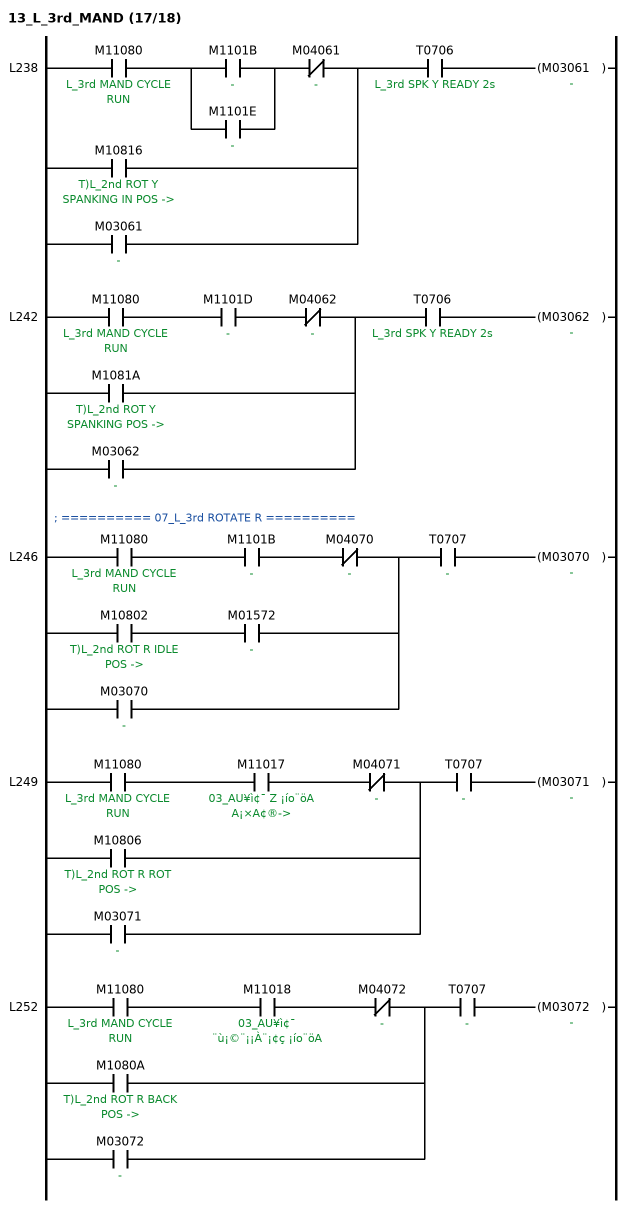
[picture p96: 13_L_3rd_MAND rungs L238-L252]
; L238
LOAD      M11080	// L_3rd MAND CYCLE RUN
LOAD      M1101B	// -
OR        M1101E	// -
AND LOAD
AND NOT   M04061	// -
OR        M10816	// T)L_2nd ROT Y SPANKING IN POS ->
OR        M03061	// -
AND       T0706	// L_3rd SPK Y READY 2s
OUT       M03061	// -
; L242
LOAD      M11080	// L_3rd MAND CYCLE RUN
AND       M1101D	// -
AND NOT   M04062	// -
OR        M1081A	// T)L_2nd ROT Y SPANKING POS ->
OR        M03062	// -
AND       T0706	// L_3rd SPK Y READY 2s
OUT       M03062	// -
// ========== 07_L_3rd ROTATE R ==========
; L246
LOAD      M11080	// L_3rd MAND CYCLE RUN
AND       M1101B	// -
AND NOT   M04070	// -
LOAD      M10802	// T)L_2nd ROT R IDLE POS ->
AND       M01572	// -
OR LOAD
OR        M03070	// -
AND       T0707	// -
OUT       M03070	// -
; L249
LOAD      M11080	// L_3rd MAND CYCLE RUN
AND       M11017	// 03_AU¥ì¢¯ Z ¡ío¨öA A¡×A¢®->
AND NOT   M04071	// -
OR        M10806	// T)L_2nd ROT R ROT POS ->
OR        M03071	// -
AND       T0707	// -
OUT       M03071	// -
; L252
LOAD      M11080	// L_3rd MAND CYCLE RUN
AND       M11018	// 03_AU¥ì¢¯ ¨ù¡©¨¡¡À¨¡¢ç ¡ío¨öA
AND NOT   M04072	// -
OR        M1080A	// T)L_2nd ROT R BACK POS ->
OR        M03072	// -
AND       T0707	// -
OUT       M03072	// -

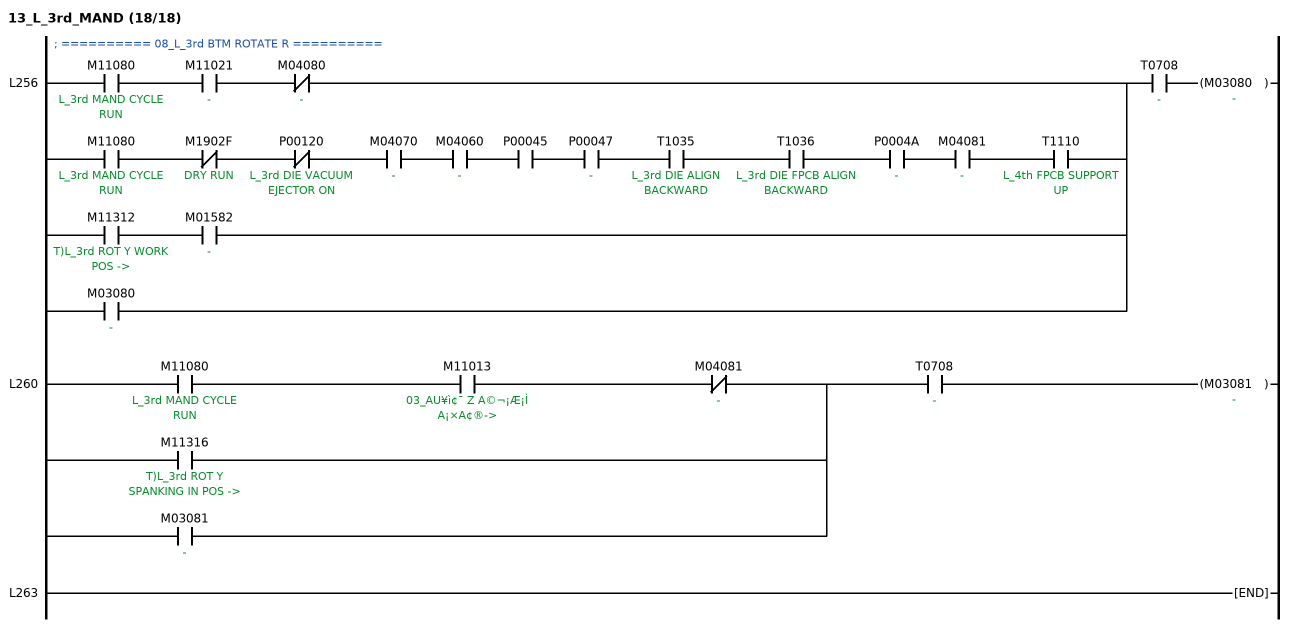
// ========== 08_L_3rd BTM ROTATE R ==========
; L256
LOAD      M11080	// L_3rd MAND CYCLE RUN
AND       M11021	// -
AND NOT   M04080	// -
LOAD      M11080	// L_3rd MAND CYCLE RUN
AND NOT   M1902F	// DRY RUN
AND NOT   P00120	// L_3rd DIE VACUUM EJECTOR ON
AND       M04070	// -
AND       M04060	// -
AND       P00045
AND       P00047	// -
AND       T1035	// L_3rd DIE ALIGN BACKWARD
AND       T1036	// L_3rd DIE FPCB ALIGN BACKWARD
AND       P0004A	// -
AND       M04081	// -
AND       T1110	// L_4th FPCB SUPPORT UP
OR LOAD
LOAD      M11312	// T)L_3rd ROT Y WORK POS ->
AND       M01582	// -
OR LOAD
OR        M03080	// -
AND       T0708	// -
OUT       M03080	// -
; L260
LOAD      M11080	// L_3rd MAND CYCLE RUN
AND       M11013	// 03_AU¥ì¢¯ Z A©¬¡Æ¡Ì A¡×A¢®->
AND NOT   M04081	// -
OR        M11316	// T)L_3rd ROT Y SPANKING IN POS ->
OR        M03081	// -
AND       T0708	// -
OUT       M03081	// -
; L263
END

PROGRAM 14_L_TOOL (task: ¨ö¨¬A¥ì CA¡¤I¡¾¡¿¡¤¡Í)

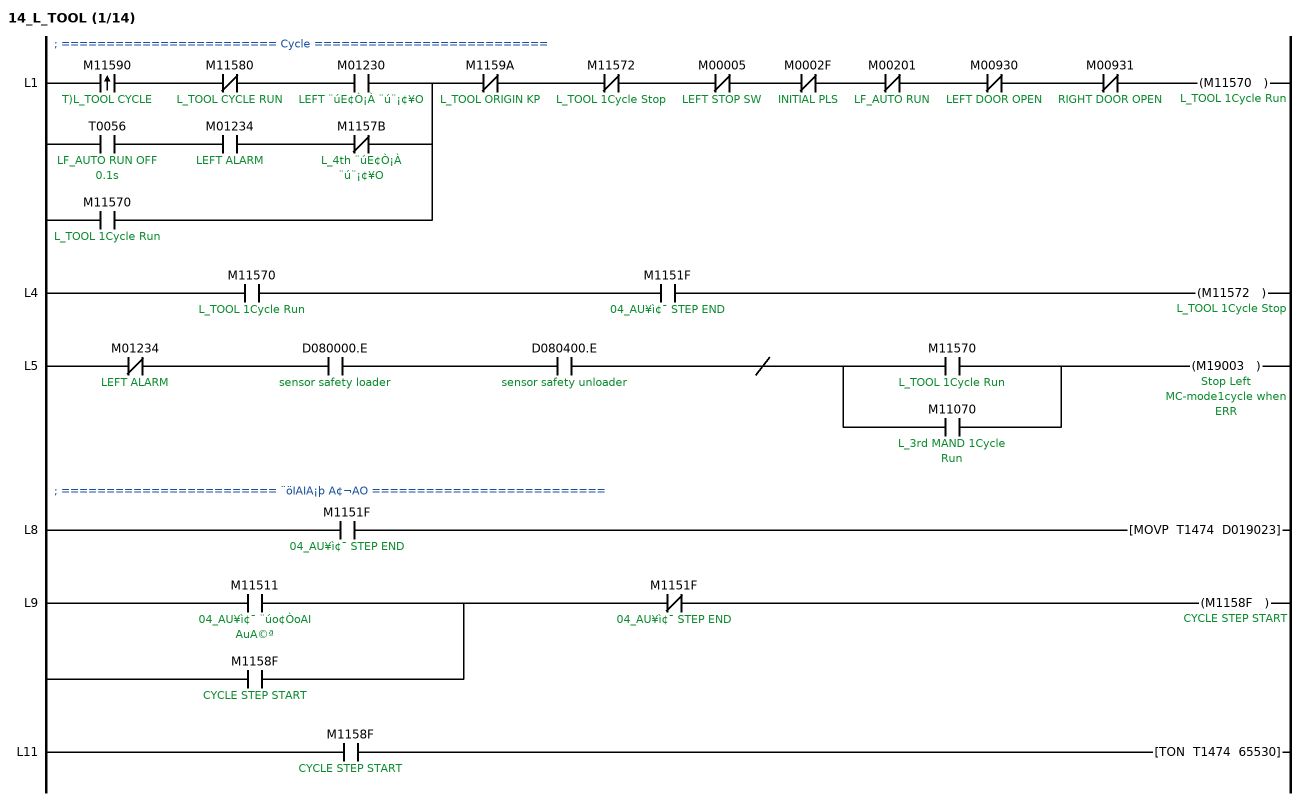
// ======================== Cycle ==========================
; L1
LOADP     M11590	// T)L_TOOL CYCLE
AND NOT   M11580	// L_TOOL CYCLE RUN
AND       M01230	// LEFT ¨úE¢Ò¡À ¨ú¨¡¢¥O
LOAD      T0056	// LF_AUTO RUN OFF 0.1s
AND       M01234	// LEFT ALARM
AND NOT   M1157B	// L_4th ¨úE¢Ò¡À ¨ú¨¡¢¥O
OR LOAD
OR        M11570	// L_TOOL 1Cycle Run
AND NOT   M1159A	// L_TOOL ORIGIN KP
AND NOT   M11572	// L_TOOL 1Cycle Stop
AND NOT   M00005	// LEFT STOP SW
AND NOT   M0002F	// INITIAL PLS
AND NOT   M00201	// LF_AUTO RUN
AND NOT   M00930	// LEFT DOOR OPEN
AND NOT   M00931	// RIGHT DOOR OPEN
OUT       M11570	// L_TOOL 1Cycle Run
; L4
LOAD      M11570	// L_TOOL 1Cycle Run
AND       M1151F	// 04_AU¥ì¢¯ STEP END
OUT       M11572	// L_TOOL 1Cycle Stop
; L5
LOAD NOT  M01234	// LEFT ALARM
AND       D080000.E	// sensor safety loader
AND       D080400.E	// sensor safety unloader
NOT
LOAD      M11570	// L_TOOL 1Cycle Run
OR        M11070	// L_3rd MAND 1Cycle Run
AND LOAD
OUT       M19003	// Stop Left MC-mode1cycle when ERR
// ======================== ¨öIAIA¡þ A¢¬AO ==========================
; L8
LOAD      M1151F	// 04_AU¥ì¢¯ STEP END
MOVP      T1474 D019023
; L9
LOAD      M11511	// 04_AU¥ì¢¯ ¨úo¢ÒoAI AuA©ª
OR        M1158F	// CYCLE STEP START
AND NOT   M1151F	// 04_AU¥ì¢¯ STEP END
OUT       M1158F	// CYCLE STEP START
; L11
LOAD      M1158F	// CYCLE STEP START
TON       T1474 65530

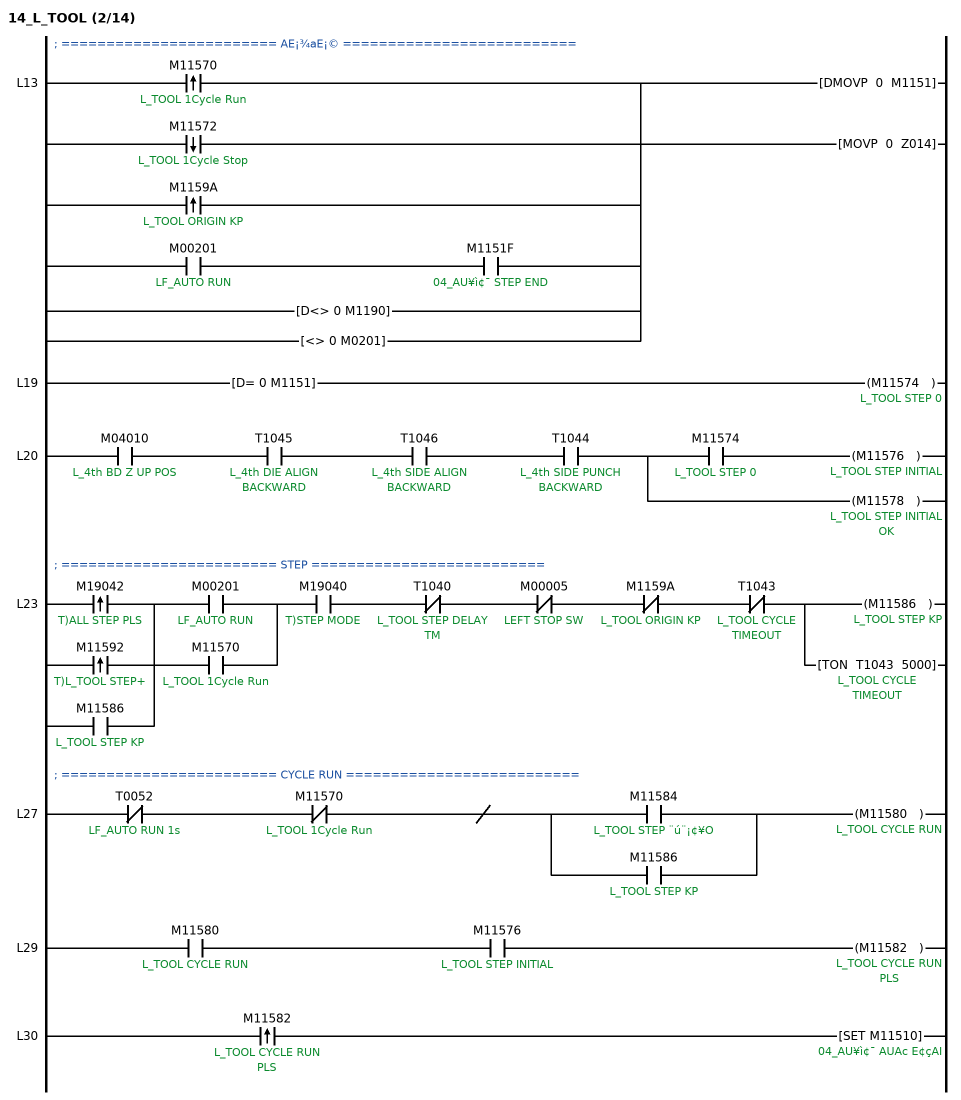
// ======================== AE¡¾aE¡© ==========================
; L13
LOADP     M11570	// L_TOOL 1Cycle Run
ORN       M11572	// L_TOOL 1Cycle Stop
ORP       M1159A	// L_TOOL ORIGIN KP
LOAD      M00201	// LF_AUTO RUN
AND       M1151F	// 04_AU¥ì¢¯ STEP END
OR LOAD
ORD<>     0 M1190
OR<>      0 M0201
DMOVP     0 M1151
MOVP      0 Z014
; L19
LOADD=    0 M1151
OUT       M11574	// L_TOOL STEP 0
; L20
LOAD      M04010	// L_4th BD Z UP POS
AND       T1045	// L_4th DIE ALIGN BACKWARD
AND       T1046	// L_4th SIDE ALIGN BACKWARD
AND       T1044	// L_4th SIDE PUNCH BACKWARD
MPUSH
AND       M11574	// L_TOOL STEP 0
OUT       M11576	// L_TOOL STEP INITIAL
MPOP
OUT       M11578	// L_TOOL STEP INITIAL OK
// ======================== STEP ==========================
; L23
LOADP     M19042	// T)ALL STEP PLS
ORP       M11592	// T)L_TOOL STEP+
OR        M11586	// L_TOOL STEP KP
LOAD      M00201	// LF_AUTO RUN
OR        M11570	// L_TOOL 1Cycle Run
AND LOAD
AND       M19040	// T)STEP MODE
AND NOT   T1040	// L_TOOL STEP DELAY TM
AND NOT   M00005	// LEFT STOP SW
AND NOT   M1159A	// L_TOOL ORIGIN KP
AND NOT   T1043	// L_TOOL CYCLE TIMEOUT
OUT       M11586	// L_TOOL STEP KP
TON       T1043 5000	// L_TOOL CYCLE TIMEOUT
// ======================== CYCLE RUN ==========================
; L27
LOAD NOT  T0052	// LF_AUTO RUN 1s
AND NOT   M11570	// L_TOOL 1Cycle Run
NOT
LOAD      M11584	// L_TOOL STEP ¨ú¨¡¢¥O
OR        M11586	// L_TOOL STEP KP
AND LOAD
OUT       M11580	// L_TOOL CYCLE RUN
; L29
LOAD      M11580	// L_TOOL CYCLE RUN
AND       M11576	// L_TOOL STEP INITIAL
OUT       M11582	// L_TOOL CYCLE RUN PLS
; L30
LOADP     M11582	// L_TOOL CYCLE RUN PLS
SET       M11510	// 04_AU¥ì¢¯ AUAc E¢çAI

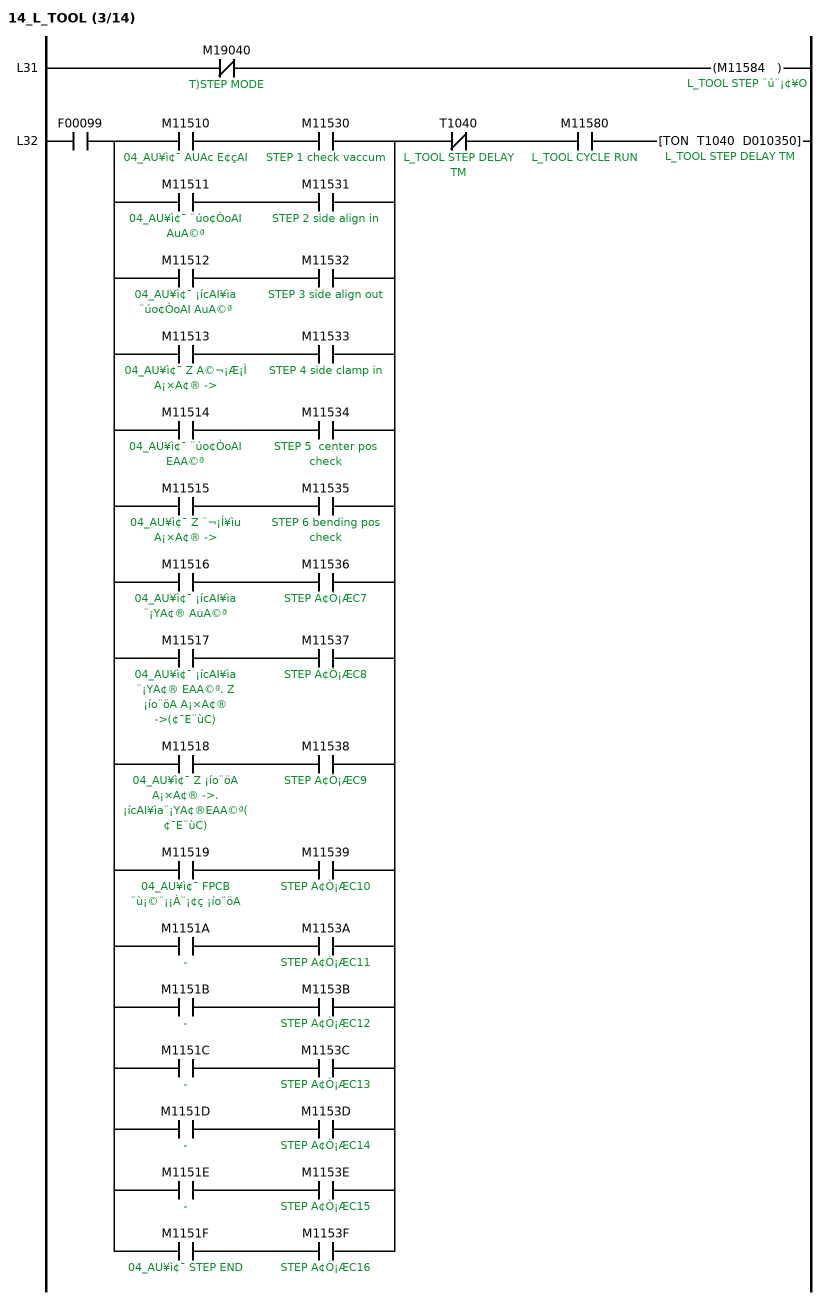
; L31
LOAD NOT  M19040	// T)STEP MODE
OUT       M11584	// L_TOOL STEP ¨ú¨¡¢¥O
; L32
LOAD      F00099
LOAD      M11510	// 04_AU¥ì¢¯ AUAc E¢çAI
AND       M11530	// STEP 1 check vaccum
LOAD      M11511	// 04_AU¥ì¢¯ ¨úo¢ÒoAI AuA©ª
AND       M11531	// STEP 2 side align in
OR LOAD
LOAD      M11512	// 04_AU¥ì¢¯ ¡ícAI¥ìa ¨úo¢ÒoAI AuA©ª
AND       M11532	// STEP 3 side align out
OR LOAD
LOAD      M11513	// 04_AU¥ì¢¯ Z A©¬¡Æ¡Ì A¡×A¢® ->
AND       M11533	// STEP 4 side clamp in
OR LOAD
LOAD      M11514	// 04_AU¥ì¢¯ ¨úo¢ÒoAI EAA©ª
AND       M11534	// STEP 5  center pos check
OR LOAD
LOAD      M11515	// 04_AU¥ì¢¯ Z ¨¬¡Í¥ìu A¡×A¢® ->
AND       M11535	// STEP 6 bending pos check
OR LOAD
LOAD      M11516	// 04_AU¥ì¢¯ ¡ícAI¥ìa ¨¡YA¢® AuA©ª
AND       M11536	// STEP A¢Ò¡ÆC7
OR LOAD
LOAD      M11517	// 04_AU¥ì¢¯ ¡ícAI¥ìa ¨¡YA¢® EAA©ª. Z ¡ío¨öA A¡×A¢® ->(¢¯E¨ùC)
AND       M11537	// STEP A¢Ò¡ÆC8
OR LOAD
LOAD      M11518	// 04_AU¥ì¢¯ Z ¡ío¨öA A¡×A¢® ->. ¡ícAI¥ìa¨¡YA¢®EAA©ª(¢¯E¨ùC)
AND       M11538	// STEP A¢Ò¡ÆC9
OR LOAD
LOAD      M11519	// 04_AU¥ì¢¯ FPCB ¨ù¡©¨¡¡À¨¡¢ç ¡ío¨öA
AND       M11539	// STEP A¢Ò¡ÆC10
OR LOAD
LOAD      M1151A	// -
AND       M1153A	// STEP A¢Ò¡ÆC11
OR LOAD
LOAD      M1151B	// -
AND       M1153B	// STEP A¢Ò¡ÆC12
OR LOAD
LOAD      M1151C	// -
AND       M1153C	// STEP A¢Ò¡ÆC13
OR LOAD
LOAD      M1151D	// -
AND       M1153D	// STEP A¢Ò¡ÆC14
OR LOAD
LOAD      M1151E	// -
AND       M1153E	// STEP A¢Ò¡ÆC15
OR LOAD
LOAD      M1151F	// 04_AU¥ì¢¯ STEP END
AND       M1153F	// STEP A¢Ò¡ÆC16
OR LOAD
AND LOAD
AND NOT   T1040	// L_TOOL STEP DELAY TM
AND       M11580	// L_TOOL CYCLE RUN
TON       T1040 D010350	// L_TOOL STEP DELAY TM

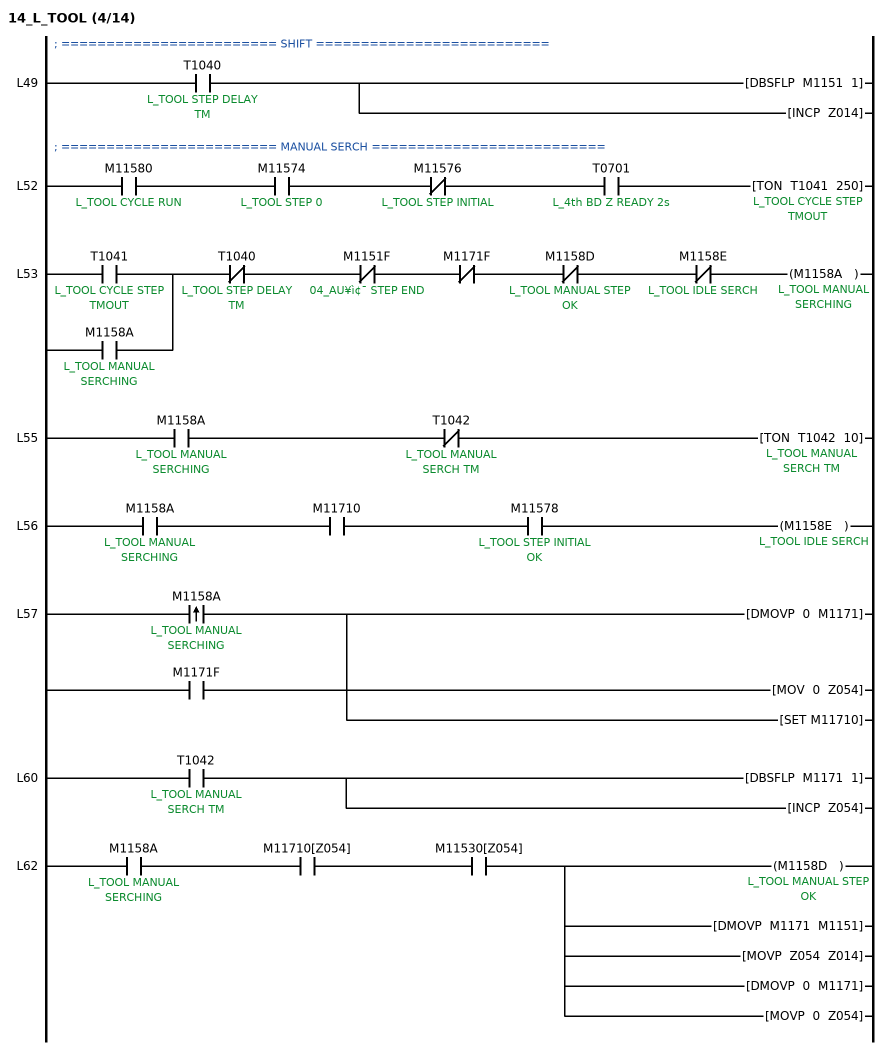
// ======================== SHIFT ==========================
; L49
LOAD      T1040	// L_TOOL STEP DELAY TM
DBSFLP    M1151 1
INCP      Z014
// ======================== MANUAL SERCH ==========================
; L52
LOAD      M11580	// L_TOOL CYCLE RUN
AND       M11574	// L_TOOL STEP 0
AND NOT   M11576	// L_TOOL STEP INITIAL
AND       T0701	// L_4th BD Z READY 2s
TON       T1041 250	// L_TOOL CYCLE STEP TMOUT
; L53
LOAD      T1041	// L_TOOL CYCLE STEP TMOUT
OR        M1158A	// L_TOOL MANUAL SERCHING
AND NOT   T1040	// L_TOOL STEP DELAY TM
AND NOT   M1151F	// 04_AU¥ì¢¯ STEP END
AND NOT   M1171F
AND NOT   M1158D	// L_TOOL MANUAL STEP OK
AND NOT   M1158E	// L_TOOL IDLE SERCH
OUT       M1158A	// L_TOOL MANUAL SERCHING
; L55
LOAD      M1158A	// L_TOOL MANUAL SERCHING
AND NOT   T1042	// L_TOOL MANUAL SERCH TM
TON       T1042 10	// L_TOOL MANUAL SERCH TM
; L56
LOAD      M1158A	// L_TOOL MANUAL SERCHING
AND       M11710
AND       M11578	// L_TOOL STEP INITIAL OK
OUT       M1158E	// L_TOOL IDLE SERCH
; L57
LOADP     M1158A	// L_TOOL MANUAL SERCHING
OR        M1171F
DMOVP     0 M1171
MOV       0 Z054
SET       M11710
; L60
LOAD      T1042	// L_TOOL MANUAL SERCH TM
DBSFLP    M1171 1
INCP      Z054
; L62
LOAD      M1158A	// L_TOOL MANUAL SERCHING
AND       M11710[Z054]
AND       M11530[Z054]
OUT       M1158D	// L_TOOL MANUAL STEP OK
DMOVP     M1171 M1151
MOVP      Z054 Z014
DMOVP     0 M1171
MOVP      0 Z054

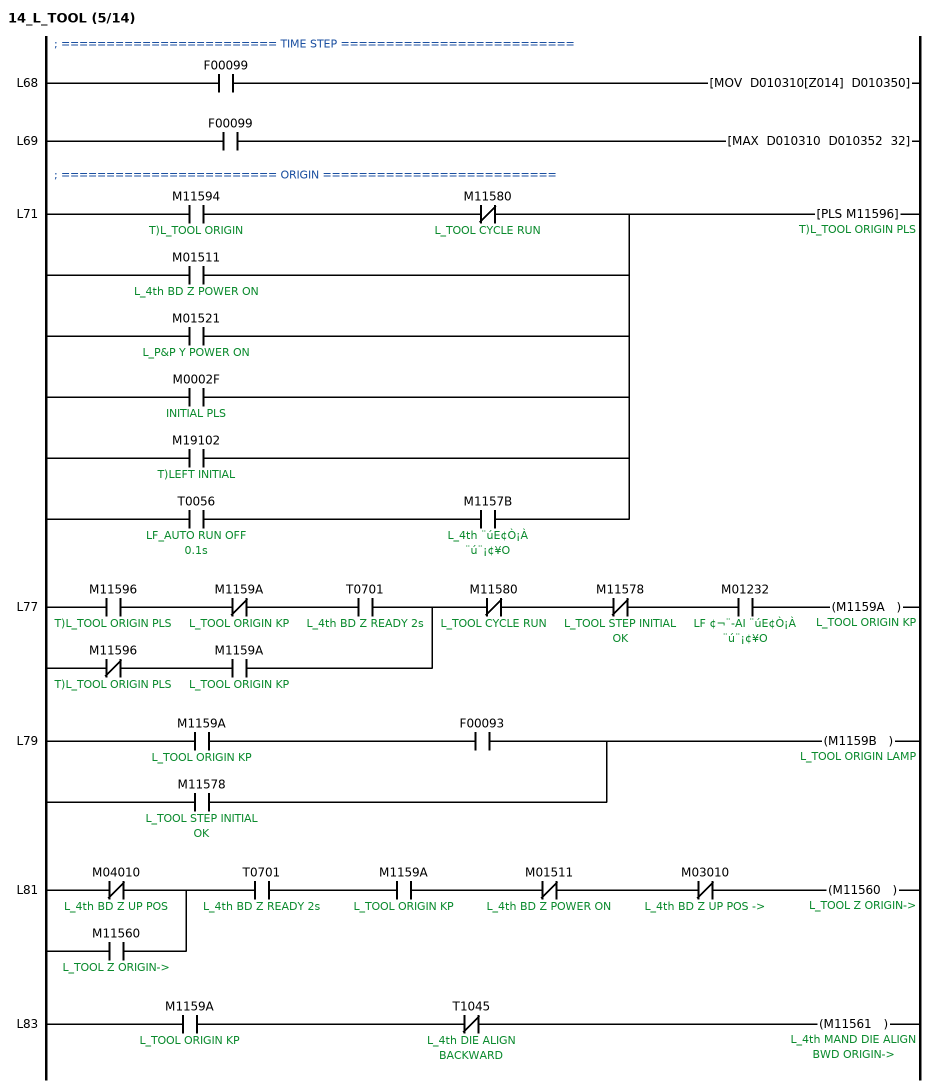
// ======================== TIME STEP ==========================
; L68
LOAD      F00099
MOV       D010310[Z014] D010350
; L69
LOAD      F00099
MAX       D010310 D010352 32
// ======================== ORIGIN ==========================
; L71
LOAD      M11594	// T)L_TOOL ORIGIN
AND NOT   M11580	// L_TOOL CYCLE RUN
OR        M01511	// L_4th BD Z POWER ON
OR        M01521	// L_P&P Y POWER ON
OR        M0002F	// INITIAL PLS
OR        M19102	// T)LEFT INITIAL
LOAD      T0056	// LF_AUTO RUN OFF 0.1s
AND       M1157B	// L_4th ¨úE¢Ò¡À ¨ú¨¡¢¥O
OR LOAD
OUTP      M11596	// T)L_TOOL ORIGIN PLS
; L77
LOAD      M11596	// T)L_TOOL ORIGIN PLS
AND NOT   M1159A	// L_TOOL ORIGIN KP
AND       T0701	// L_4th BD Z READY 2s
LOAD NOT  M11596	// T)L_TOOL ORIGIN PLS
AND       M1159A	// L_TOOL ORIGIN KP
OR LOAD
AND NOT   M11580	// L_TOOL CYCLE RUN
AND NOT   M11578	// L_TOOL STEP INITIAL OK
AND       M01232	// LF ¢¬¨­AI ¨úE¢Ò¡À ¨ú¨¡¢¥O
OUT       M1159A	// L_TOOL ORIGIN KP
; L79
LOAD      M1159A	// L_TOOL ORIGIN KP
AND       F00093
OR        M11578	// L_TOOL STEP INITIAL OK
OUT       M1159B	// L_TOOL ORIGIN LAMP
; L81
LOAD NOT  M04010	// L_4th BD Z UP POS
OR        M11560	// L_TOOL Z ORIGIN->
AND       T0701	// L_4th BD Z READY 2s
AND       M1159A	// L_TOOL ORIGIN KP
AND NOT   M01511	// L_4th BD Z POWER ON
AND NOT   M03010	// L_4th BD Z UP POS ->
OUT       M11560	// L_TOOL Z ORIGIN->
; L83
LOAD      M1159A	// L_TOOL ORIGIN KP
AND NOT   T1045	// L_4th DIE ALIGN BACKWARD
OUT       M11561	// L_4th MAND DIE ALIGN BWD ORIGIN->

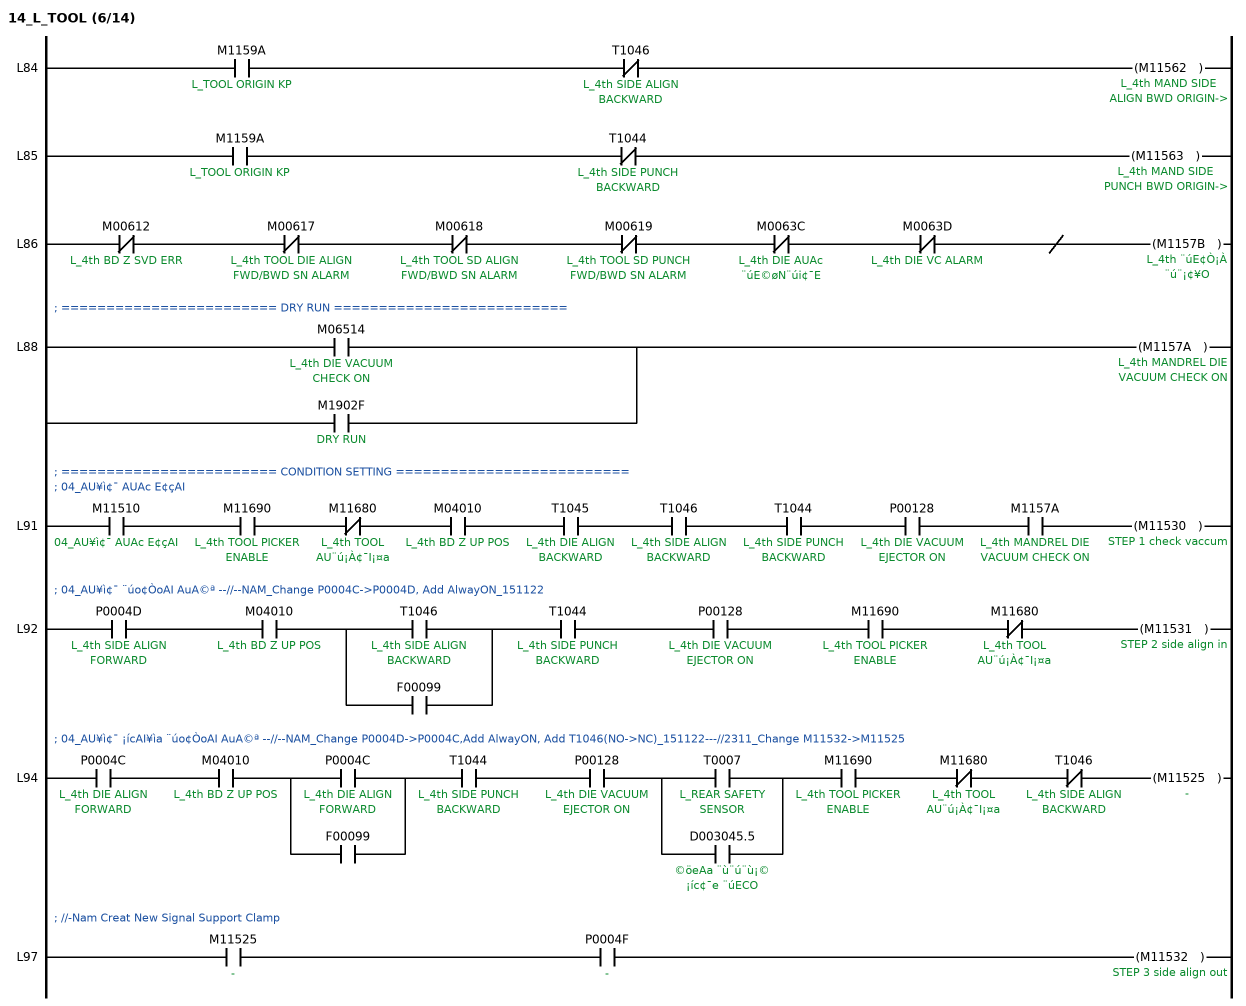
; L84
LOAD      M1159A	// L_TOOL ORIGIN KP
AND NOT   T1046	// L_4th SIDE ALIGN BACKWARD
OUT       M11562	// L_4th MAND SIDE ALIGN BWD ORIGIN->
; L85
LOAD      M1159A	// L_TOOL ORIGIN KP
AND NOT   T1044	// L_4th SIDE PUNCH BACKWARD
OUT       M11563	// L_4th MAND SIDE PUNCH BWD ORIGIN->
; L86
LOAD NOT  M00612	// L_4th BD Z SVD ERR
AND NOT   M00617	// L_4th TOOL DIE ALIGN FWD/BWD SN ALARM
AND NOT   M00618	// L_4th TOOL SD ALIGN FWD/BWD SN ALARM
AND NOT   M00619	// L_4th TOOL SD PUNCH FWD/BWD SN ALARM
AND NOT   M0063C	// L_4th DIE AUAc ¨úE©øN¨úi¢¯E
AND NOT   M0063D	// L_4th DIE VC ALARM
NOT
OUT       M1157B	// L_4th ¨úE¢Ò¡À ¨ú¨¡¢¥O
// ======================== DRY RUN ==========================
; L88
LOAD      M06514	// L_4th DIE VACUUM CHECK ON
OR        M1902F	// DRY RUN
OUT       M1157A	// L_4th MANDREL DIE VACUUM CHECK ON
// ======================== CONDITION SETTING ==========================
; L91
LOAD      M11510	// 04_AU¥ì¢¯ AUAc E¢çAI
AND       M11690	// L_4th TOOL PICKER ENABLE
AND NOT   M11680	// L_4th TOOL AU¨ú¡À¢¯I¡¤a
AND       M04010	// L_4th BD Z UP POS
AND       T1045	// L_4th DIE ALIGN BACKWARD
AND       T1046	// L_4th SIDE ALIGN BACKWARD
AND       T1044	// L_4th SIDE PUNCH BACKWARD
AND       P00128	// L_4th DIE VACUUM EJECTOR ON
AND       M1157A	// L_4th MANDREL DIE VACUUM CHECK ON
OUT       M11530	// STEP 1 check vaccum
// output comment: 04_AU¥ì¢¯ AUAc E¢çAI
; L92
LOAD      P0004D	// L_4th SIDE ALIGN FORWARD
AND       M04010	// L_4th BD Z UP POS
LOAD      T1046	// L_4th SIDE ALIGN BACKWARD
OR        F00099
AND LOAD
AND       T1044	// L_4th SIDE PUNCH BACKWARD
AND       P00128	// L_4th DIE VACUUM EJECTOR ON
AND       M11690	// L_4th TOOL PICKER ENABLE
AND NOT   M11680	// L_4th TOOL AU¨ú¡À¢¯I¡¤a
OUT       M11531	// STEP 2 side align in
// output comment: 04_AU¥ì¢¯ ¨úo¢ÒoAI AuA©ª --//--NAM_Change P0004C->P0004D, Add AlwayON_151122
; L94
LOAD      P0004C	// L_4th DIE ALIGN FORWARD
AND       M04010	// L_4th BD Z UP POS
LOAD      P0004C	// L_4th DIE ALIGN FORWARD
OR        F00099
AND LOAD
AND       T1044	// L_4th SIDE PUNCH BACKWARD
AND       P00128	// L_4th DIE VACUUM EJECTOR ON
LOAD      T0007	// L_REAR SAFETY SENSOR
OR        D003045.5	// ©öeAa ¨ù¨ú¨ù¡© ¡íc¢¯e ¨úECO
AND LOAD
AND       M11690	// L_4th TOOL PICKER ENABLE
AND NOT   M11680	// L_4th TOOL AU¨ú¡À¢¯I¡¤a
AND NOT   T1046	// L_4th SIDE ALIGN BACKWARD
OUT       M11525	// -
// output comment: 04_AU¥ì¢¯ ¡ícAI¥ìa ¨úo¢ÒoAI AuA©ª --//--NAM_Change P0004D->P0004C,Add AlwayON, Add T1046(NO->NC)_151122---//2311_Change M11532->M11525
// //-Nam Creat New Signal Support Clamp
; L97
LOAD      M11525	// -
AND       P0004F	// -
OUT       M11532	// STEP 3 side align out

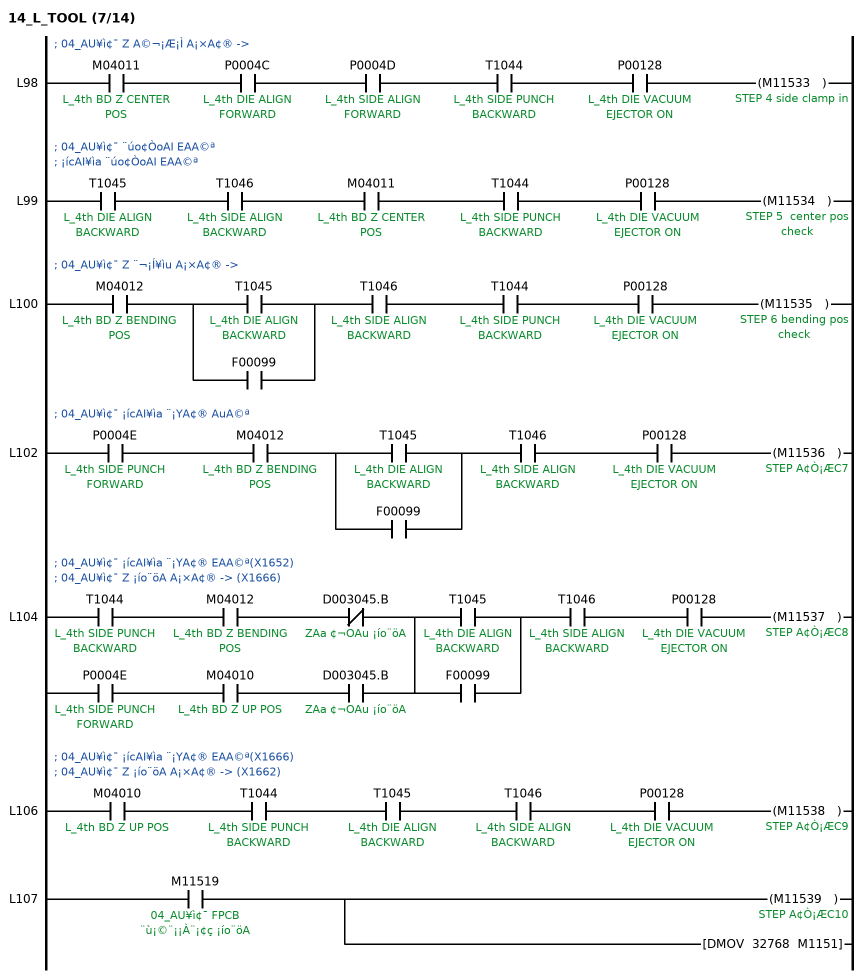
; L98
LOAD      M04011	// L_4th BD Z CENTER POS
AND       P0004C	// L_4th DIE ALIGN FORWARD
AND       P0004D	// L_4th SIDE ALIGN FORWARD
AND       T1044	// L_4th SIDE PUNCH BACKWARD
AND       P00128	// L_4th DIE VACUUM EJECTOR ON
OUT       M11533	// STEP 4 side clamp in
// output comment: 04_AU¥ì¢¯ Z A©¬¡Æ¡Ì A¡×A¢® ->
; L99
LOAD      T1045	// L_4th DIE ALIGN BACKWARD
AND       T1046	// L_4th SIDE ALIGN BACKWARD
AND       M04011	// L_4th BD Z CENTER POS
AND       T1044	// L_4th SIDE PUNCH BACKWARD
AND       P00128	// L_4th DIE VACUUM EJECTOR ON
OUT       M11534	// STEP 5  center pos check
// output comment: 04_AU¥ì¢¯ ¨úo¢ÒoAI EAA©ª ¡ícAI¥ìa ¨úo¢ÒoAI EAA©ª
; L100
LOAD      M04012	// L_4th BD Z BENDING POS
LOAD      T1045	// L_4th DIE ALIGN BACKWARD
OR        F00099
AND LOAD
AND       T1046	// L_4th SIDE ALIGN BACKWARD
AND       T1044	// L_4th SIDE PUNCH BACKWARD
AND       P00128	// L_4th DIE VACUUM EJECTOR ON
OUT       M11535	// STEP 6 bending pos check
// output comment: 04_AU¥ì¢¯ Z ¨¬¡Í¥ìu A¡×A¢® ->
; L102
LOAD      P0004E	// L_4th SIDE PUNCH FORWARD
AND       M04012	// L_4th BD Z BENDING POS
LOAD      T1045	// L_4th DIE ALIGN BACKWARD
OR        F00099
AND LOAD
AND       T1046	// L_4th SIDE ALIGN BACKWARD
AND       P00128	// L_4th DIE VACUUM EJECTOR ON
OUT       M11536	// STEP A¢Ò¡ÆC7
// output comment: 04_AU¥ì¢¯ ¡ícAI¥ìa ¨¡YA¢® AuA©ª
; L104
LOAD      T1044	// L_4th SIDE PUNCH BACKWARD
AND       M04012	// L_4th BD Z BENDING POS
AND NOT   D003045.B	// ZAa ¢¬OAu ¡ío¨öA
LOAD      P0004E	// L_4th SIDE PUNCH FORWARD
AND       M04010	// L_4th BD Z UP POS
AND       D003045.B	// ZAa ¢¬OAu ¡ío¨öA
OR LOAD
LOAD      T1045	// L_4th DIE ALIGN BACKWARD
OR        F00099
AND LOAD
AND       T1046	// L_4th SIDE ALIGN BACKWARD
AND       P00128	// L_4th DIE VACUUM EJECTOR ON
OUT       M11537	// STEP A¢Ò¡ÆC8
// output comment: 04_AU¥ì¢¯ ¡ícAI¥ìa ¨¡YA¢® EAA©ª(X1652) 04_AU¥ì¢¯ Z ¡ío¨öA A¡×A¢® -> (X1666)
; L106
LOAD      M04010	// L_4th BD Z UP POS
AND       T1044	// L_4th SIDE PUNCH BACKWARD
AND       T1045	// L_4th DIE ALIGN BACKWARD
AND       T1046	// L_4th SIDE ALIGN BACKWARD
AND       P00128	// L_4th DIE VACUUM EJECTOR ON
OUT       M11538	// STEP A¢Ò¡ÆC9
// output comment: 04_AU¥ì¢¯ ¡ícAI¥ìa ¨¡YA¢® EAA©ª(X1666) 04_AU¥ì¢¯ Z ¡ío¨öA A¡×A¢® -> (X1662)
; L107
LOAD      M11519	// 04_AU¥ì¢¯ FPCB ¨ù¡©¨¡¡À¨¡¢ç ¡ío¨öA
OUT       M11539	// STEP A¢Ò¡ÆC10
DMOV      32768 M1151

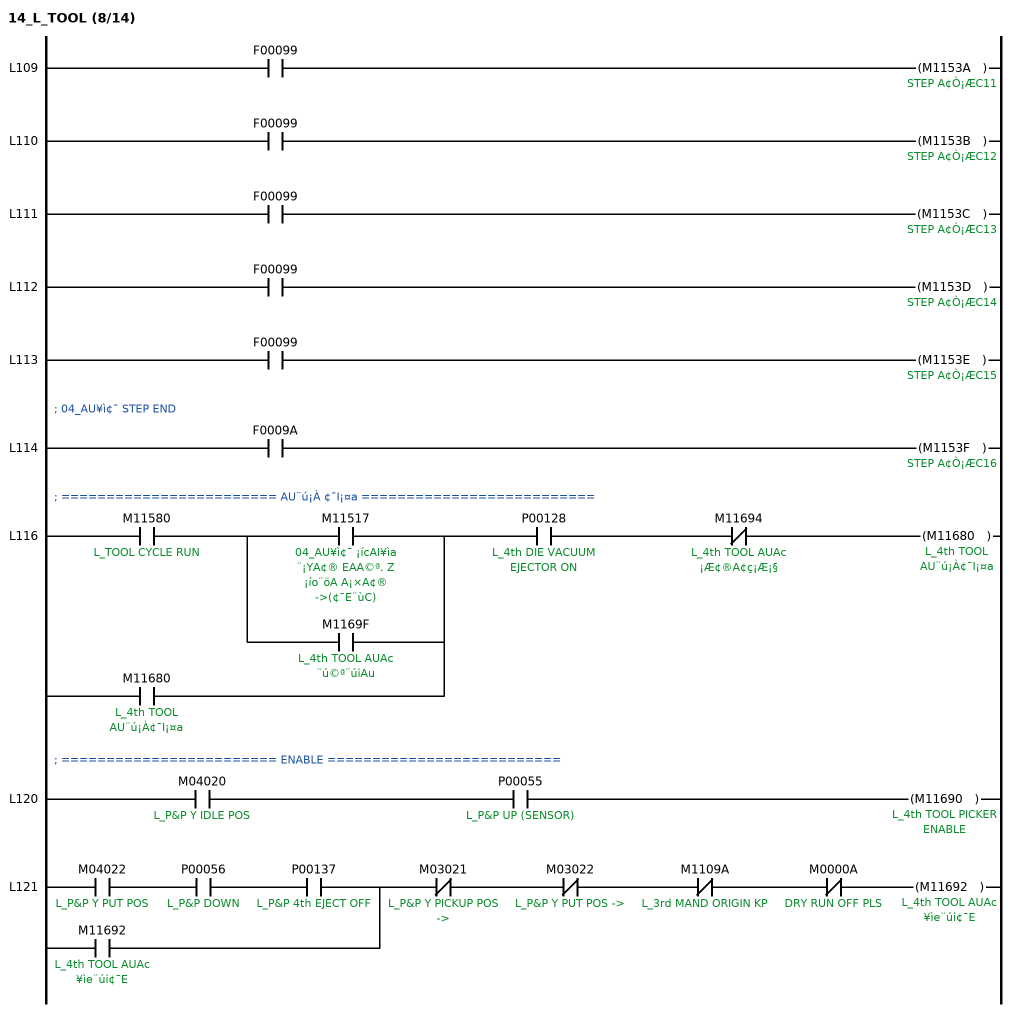
; L109
LOAD      F00099
OUT       M1153A	// STEP A¢Ò¡ÆC11
; L110
LOAD      F00099
OUT       M1153B	// STEP A¢Ò¡ÆC12
; L111
LOAD      F00099
OUT       M1153C	// STEP A¢Ò¡ÆC13
; L112
LOAD      F00099
OUT       M1153D	// STEP A¢Ò¡ÆC14
; L113
LOAD      F00099
OUT       M1153E	// STEP A¢Ò¡ÆC15
; L114
LOAD      F0009A
OUT       M1153F	// STEP A¢Ò¡ÆC16
// output comment: 04_AU¥ì¢¯ STEP END
// ======================== AU¨ú¡À ¢¯I¡¤a ==========================
; L116
LOAD      M11580	// L_TOOL CYCLE RUN
LOAD      M11517	// 04_AU¥ì¢¯ ¡ícAI¥ìa ¨¡YA¢® EAA©ª. Z ¡ío¨öA A¡×A¢® ->(¢¯E¨ùC)
OR        M1169F	// L_4th TOOL AUAc ¨ú©ª¨úiAu
AND LOAD
OR        M11680	// L_4th TOOL AU¨ú¡À¢¯I¡¤a
AND       P00128	// L_4th DIE VACUUM EJECTOR ON
AND NOT   M11694	// L_4th TOOL AUAc ¡Æ¢®A¢ç¡Æ¡§
OUT       M11680	// L_4th TOOL AU¨ú¡À¢¯I¡¤a
// ======================== ENABLE ==========================
; L120
LOAD      M04020	// L_P&P Y IDLE POS
AND       P00055	// L_P&P UP (SENSOR)
OUT       M11690	// L_4th TOOL PICKER ENABLE
; L121
LOAD      M04022	// L_P&P Y PUT POS
AND       P00056	// L_P&P DOWN
AND       P00137	// L_P&P 4th EJECT OFF
OR        M11692	// L_4th TOOL AUAc ¥ìe¨úi¢¯E
AND NOT   M03021	// L_P&P Y PICKUP POS ->
AND NOT   M03022	// L_P&P Y PUT POS ->
AND NOT   M1109A	// L_3rd MAND ORIGIN KP
AND NOT   M0000A	// DRY RUN OFF PLS
OUT       M11692	// L_4th TOOL AUAc ¥ìe¨úi¢¯E

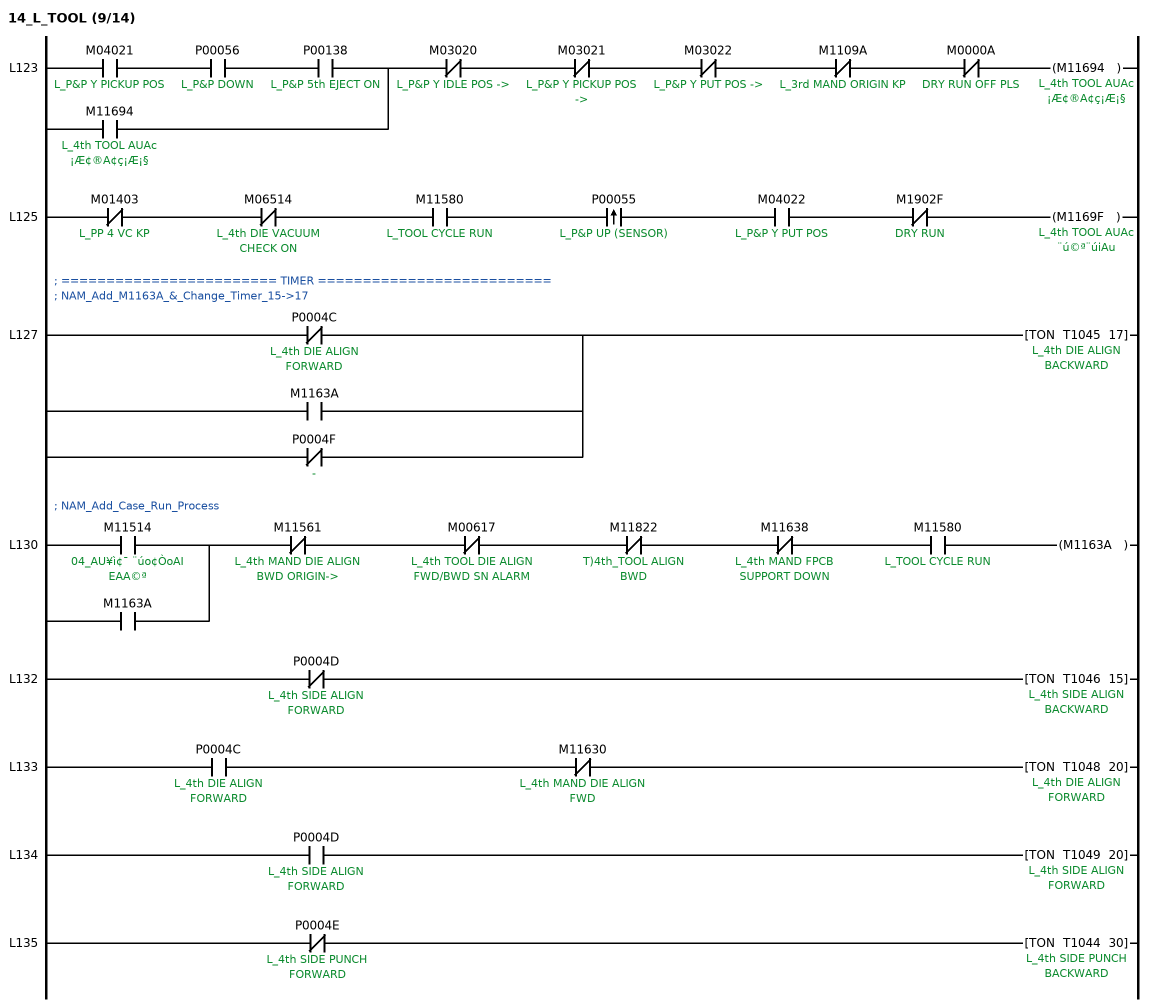
; L123
LOAD      M04021	// L_P&P Y PICKUP POS
AND       P00056	// L_P&P DOWN
AND       P00138	// L_P&P 5th EJECT ON
OR        M11694	// L_4th TOOL AUAc ¡Æ¢®A¢ç¡Æ¡§
AND NOT   M03020	// L_P&P Y IDLE POS ->
AND NOT   M03021	// L_P&P Y PICKUP POS ->
AND NOT   M03022	// L_P&P Y PUT POS ->
AND NOT   M1109A	// L_3rd MAND ORIGIN KP
AND NOT   M0000A	// DRY RUN OFF PLS
OUT       M11694	// L_4th TOOL AUAc ¡Æ¢®A¢ç¡Æ¡§
; L125
LOAD NOT  M01403	// L_PP 4 VC KP
AND NOT   M06514	// L_4th DIE VACUUM CHECK ON
AND       M11580	// L_TOOL CYCLE RUN
ANDP      P00055	// L_P&P UP (SENSOR)
AND       M04022	// L_P&P Y PUT POS
AND NOT   M1902F	// DRY RUN
OUT       M1169F	// L_4th TOOL AUAc ¨ú©ª¨úiAu
// ======================== TIMER ==========================
; L127
LOAD NOT  P0004C	// L_4th DIE ALIGN FORWARD
OR        M1163A
OR NOT    P0004F	// -
TON       T1045 17	// L_4th DIE ALIGN BACKWARD
// output comment: NAM_Add_M1163A_&_Change_Timer_15->17
; L130
LOAD      M11514	// 04_AU¥ì¢¯ ¨úo¢ÒoAI EAA©ª
OR        M1163A
AND NOT   M11561	// L_4th MAND DIE ALIGN BWD ORIGIN->
AND NOT   M00617	// L_4th TOOL DIE ALIGN FWD/BWD SN ALARM
AND NOT   M11822	// T)4th_TOOL ALIGN BWD
AND NOT   M11638	// L_4th MAND FPCB SUPPORT DOWN
AND       M11580	// L_TOOL CYCLE RUN
OUT       M1163A
// output comment: NAM_Add_Case_Run_Process
; L132
LOAD NOT  P0004D	// L_4th SIDE ALIGN FORWARD
TON       T1046 15	// L_4th SIDE ALIGN BACKWARD
; L133
LOAD      P0004C	// L_4th DIE ALIGN FORWARD
AND NOT   M11630	// L_4th MAND DIE ALIGN FWD
TON       T1048 20	// L_4th DIE ALIGN FORWARD
// output comment: 
; L134
LOAD      P0004D	// L_4th SIDE ALIGN FORWARD
TON       T1049 20	// L_4th SIDE ALIGN FORWARD
; L135
LOAD NOT  P0004E	// L_4th SIDE PUNCH FORWARD
TON       T1044 30	// L_4th SIDE PUNCH BACKWARD

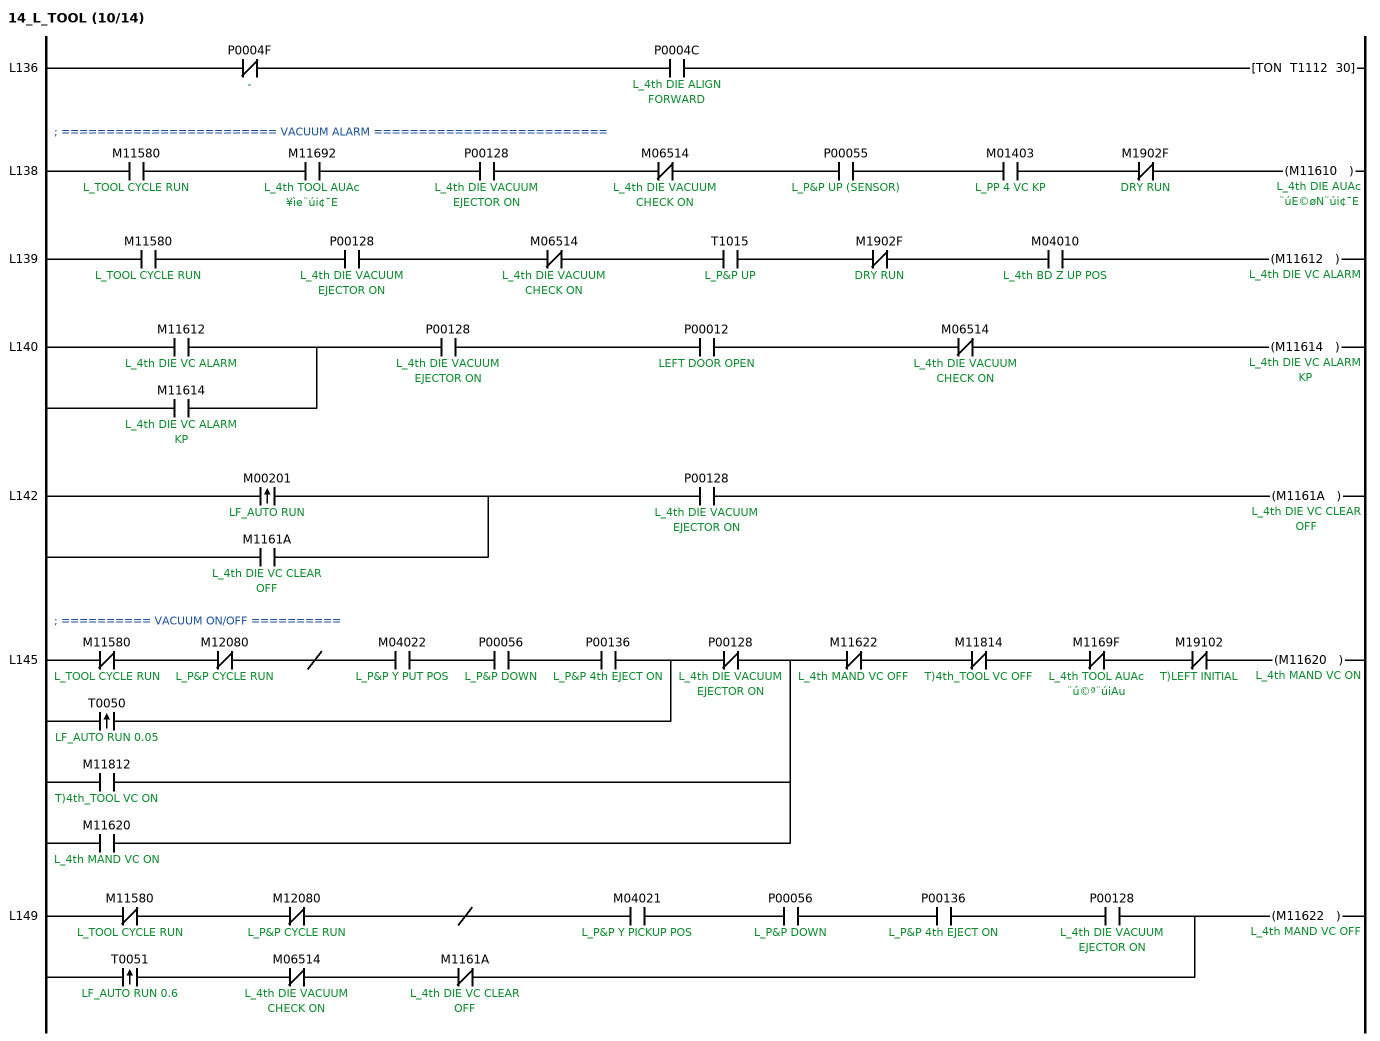
; L136
LOAD NOT  P0004F	// -
AND       P0004C	// L_4th DIE ALIGN FORWARD
TON       T1112 30
// ======================== VACUUM ALARM ==========================
; L138
LOAD      M11580	// L_TOOL CYCLE RUN
AND       M11692	// L_4th TOOL AUAc ¥ìe¨úi¢¯E
AND       P00128	// L_4th DIE VACUUM EJECTOR ON
AND NOT   M06514	// L_4th DIE VACUUM CHECK ON
AND       P00055	// L_P&P UP (SENSOR)
AND       M01403	// L_PP 4 VC KP
AND NOT   M1902F	// DRY RUN
OUT       M11610	// L_4th DIE AUAc ¨úE©øN¨úi¢¯E
; L139
LOAD      M11580	// L_TOOL CYCLE RUN
AND       P00128	// L_4th DIE VACUUM EJECTOR ON
AND NOT   M06514	// L_4th DIE VACUUM CHECK ON
AND       T1015	// L_P&P UP
AND NOT   M1902F	// DRY RUN
AND       M04010	// L_4th BD Z UP POS
OUT       M11612	// L_4th DIE VC ALARM
; L140
LOAD      M11612	// L_4th DIE VC ALARM
OR        M11614	// L_4th DIE VC ALARM KP
AND       P00128	// L_4th DIE VACUUM EJECTOR ON
AND       P00012	// LEFT DOOR OPEN
AND NOT   M06514	// L_4th DIE VACUUM CHECK ON
OUT       M11614	// L_4th DIE VC ALARM KP
; L142
LOADP     M00201	// LF_AUTO RUN
OR        M1161A	// L_4th DIE VC CLEAR OFF
AND       P00128	// L_4th DIE VACUUM EJECTOR ON
OUT       M1161A	// L_4th DIE VC CLEAR OFF
// ========== VACUUM ON/OFF ==========
; L145
LOAD NOT  M11580	// L_TOOL CYCLE RUN
AND NOT   M12080	// L_P&P CYCLE RUN
NOT
AND       M04022	// L_P&P Y PUT POS
AND       P00056	// L_P&P DOWN
AND       P00136	// L_P&P 4th EJECT ON
ORP       T0050	// LF_AUTO RUN 0.05
AND NOT   P00128	// L_4th DIE VACUUM EJECTOR ON
OR        M11812	// T)4th_TOOL VC ON
OR        M11620	// L_4th MAND VC ON
AND NOT   M11622	// L_4th MAND VC OFF
AND NOT   M11814	// T)4th_TOOL VC OFF
AND NOT   M1169F	// L_4th TOOL AUAc ¨ú©ª¨úiAu
AND NOT   M19102	// T)LEFT INITIAL
OUT       M11620	// L_4th MAND VC ON
; L149
LOAD NOT  M11580	// L_TOOL CYCLE RUN
AND NOT   M12080	// L_P&P CYCLE RUN
NOT
AND       M04021	// L_P&P Y PICKUP POS
AND       P00056	// L_P&P DOWN
AND       P00136	// L_P&P 4th EJECT ON
AND       P00128	// L_4th DIE VACUUM EJECTOR ON
LOADP     T0051	// LF_AUTO RUN 0.6
AND NOT   M06514	// L_4th DIE VACUUM CHECK ON
AND NOT   M1161A	// L_4th DIE VC CLEAR OFF
OR LOAD
OUT       M11622	// L_4th MAND VC OFF

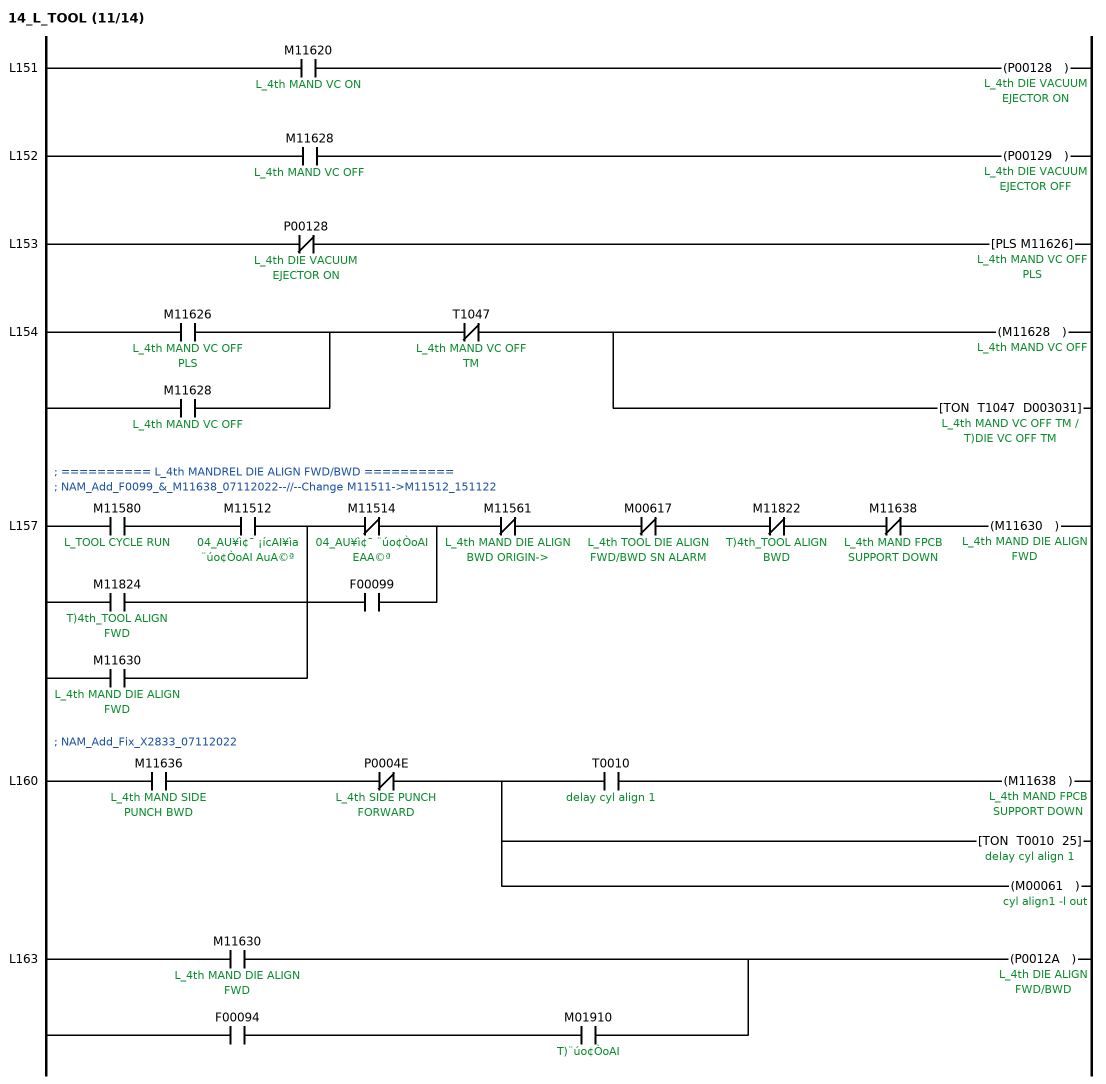
; L151
LOAD      M11620	// L_4th MAND VC ON
OUT       P00128	// L_4th DIE VACUUM EJECTOR ON
; L152
LOAD      M11628	// L_4th MAND VC OFF
OUT       P00129	// L_4th DIE VACUUM EJECTOR OFF
; L153
LOAD NOT  P00128	// L_4th DIE VACUUM EJECTOR ON
OUTP      M11626	// L_4th MAND VC OFF PLS
; L154
LOAD      M11626	// L_4th MAND VC OFF PLS
OR        M11628	// L_4th MAND VC OFF
AND NOT   T1047	// L_4th MAND VC OFF TM
OUT       M11628	// L_4th MAND VC OFF
TON       T1047 D003031	// L_4th MAND VC OFF TM / T)DIE VC OFF TM
// ========== L_4th MANDREL DIE ALIGN FWD/BWD ==========
; L157
LOAD      M11580	// L_TOOL CYCLE RUN
AND       M11512	// 04_AU¥ì¢¯ ¡ícAI¥ìa ¨úo¢ÒoAI AuA©ª
OR        M11824	// T)4th_TOOL ALIGN FWD
OR        M11630	// L_4th MAND DIE ALIGN FWD
LOAD NOT  M11514	// 04_AU¥ì¢¯ ¨úo¢ÒoAI EAA©ª
OR        F00099
AND LOAD
AND NOT   M11561	// L_4th MAND DIE ALIGN BWD ORIGIN->
AND NOT   M00617	// L_4th TOOL DIE ALIGN FWD/BWD SN ALARM
AND NOT   M11822	// T)4th_TOOL ALIGN BWD
AND NOT   M11638	// L_4th MAND FPCB SUPPORT DOWN
OUT       M11630	// L_4th MAND DIE ALIGN FWD
// output comment: NAM_Add_F0099_&_M11638_07112022--//--Change M11511->M11512_151122
; L160
LOAD      M11636	// L_4th MAND SIDE PUNCH BWD
AND NOT   P0004E	// L_4th SIDE PUNCH FORWARD
MPUSH
AND       T0010	// delay cyl align 1
OUT       M11638	// L_4th MAND FPCB SUPPORT DOWN
MPOP
TON       T0010 25	// delay cyl align 1
OUT       M00061	// cyl align1 -l out
// output comment: NAM_Add_Fix_X2833_07112022
; L163
LOAD      M11630	// L_4th MAND DIE ALIGN FWD
LOAD      F00094
AND       M01910	// T)¨úo¢ÒoAI
OR LOAD
OUT       P0012A	// L_4th DIE ALIGN FWD/BWD

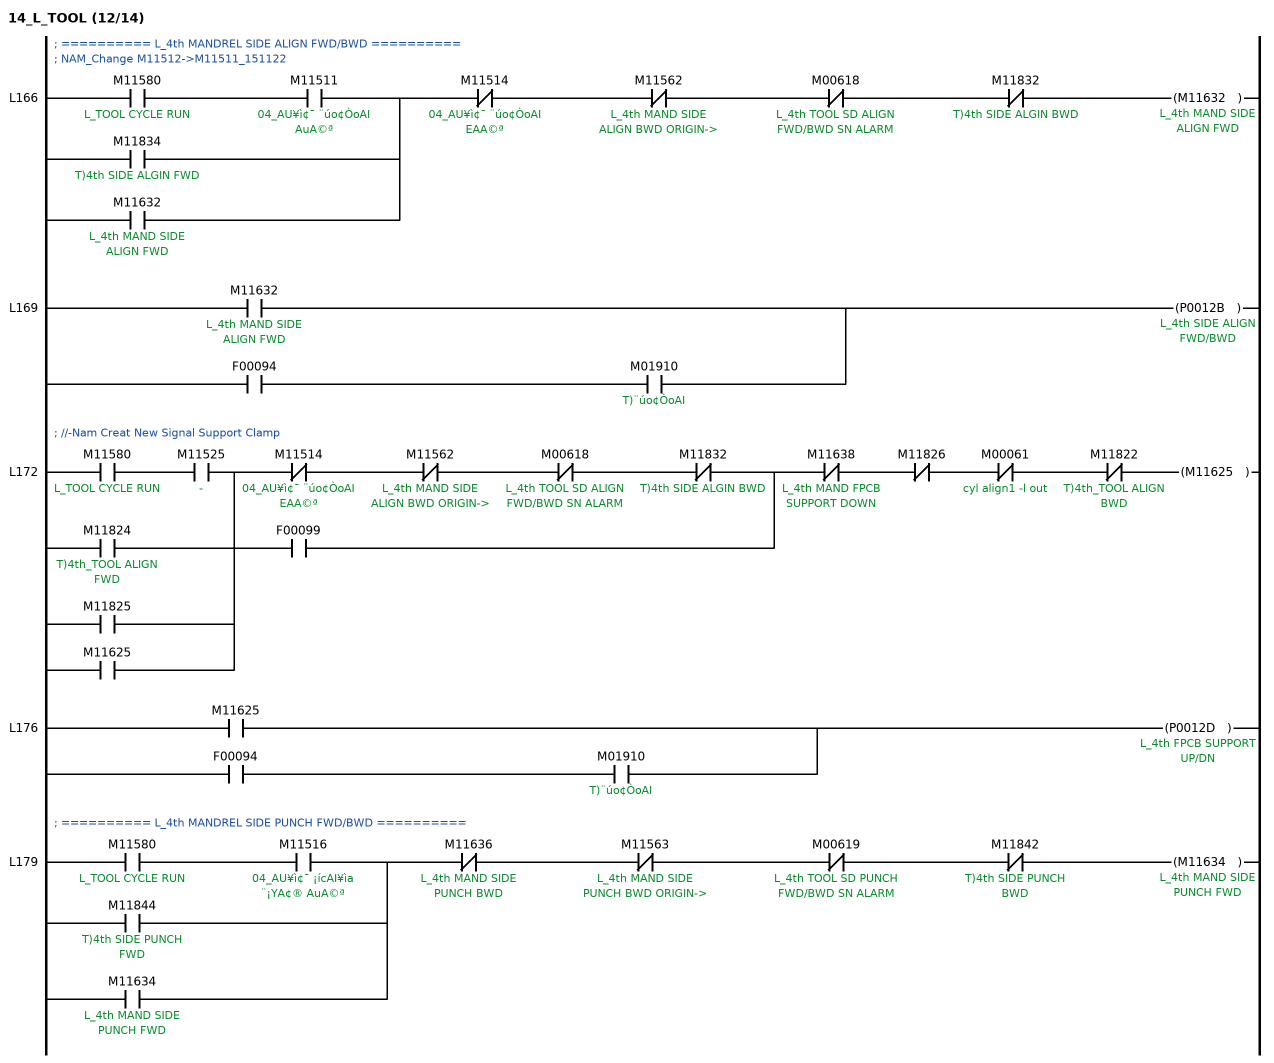
// ========== L_4th MANDREL SIDE ALIGN FWD/BWD ==========
; L166
LOAD      M11580	// L_TOOL CYCLE RUN
AND       M11511	// 04_AU¥ì¢¯ ¨úo¢ÒoAI AuA©ª
OR        M11834	// T)4th SIDE ALGIN FWD
OR        M11632	// L_4th MAND SIDE ALIGN FWD
AND NOT   M11514	// 04_AU¥ì¢¯ ¨úo¢ÒoAI EAA©ª
AND NOT   M11562	// L_4th MAND SIDE ALIGN BWD ORIGIN->
AND NOT   M00618	// L_4th TOOL SD ALIGN FWD/BWD SN ALARM
AND NOT   M11832	// T)4th SIDE ALGIN BWD
OUT       M11632	// L_4th MAND SIDE ALIGN FWD
// output comment: NAM_Change M11512->M11511_151122
; L169
LOAD      M11632	// L_4th MAND SIDE ALIGN FWD
LOAD      F00094
AND       M01910	// T)¨úo¢ÒoAI
OR LOAD
OUT       P0012B	// L_4th SIDE ALIGN FWD/BWD
// //-Nam Creat New Signal Support Clamp
; L172
LOAD      M11580	// L_TOOL CYCLE RUN
AND       M11525	// -
OR        M11824	// T)4th_TOOL ALIGN FWD
OR        M11825
OR        M11625
LOAD NOT  M11514	// 04_AU¥ì¢¯ ¨úo¢ÒoAI EAA©ª
AND NOT   M11562	// L_4th MAND SIDE ALIGN BWD ORIGIN->
AND NOT   M00618	// L_4th TOOL SD ALIGN FWD/BWD SN ALARM
AND NOT   M11832	// T)4th SIDE ALGIN BWD
OR        F00099
AND LOAD
AND NOT   M11638	// L_4th MAND FPCB SUPPORT DOWN
AND NOT   M11826
AND NOT   M00061	// cyl align1 -l out
AND NOT   M11822	// T)4th_TOOL ALIGN BWD
OUT       M11625
; L176
LOAD      M11625
LOAD      F00094
AND       M01910	// T)¨úo¢ÒoAI
OR LOAD
OUT       P0012D	// L_4th FPCB SUPPORT UP/DN
// ========== L_4th MANDREL SIDE PUNCH FWD/BWD ==========
; L179
LOAD      M11580	// L_TOOL CYCLE RUN
AND       M11516	// 04_AU¥ì¢¯ ¡ícAI¥ìa ¨¡YA¢® AuA©ª
OR        M11844	// T)4th SIDE PUNCH FWD
OR        M11634	// L_4th MAND SIDE PUNCH FWD
AND NOT   M11636	// L_4th MAND SIDE PUNCH BWD
AND NOT   M11563	// L_4th MAND SIDE PUNCH BWD ORIGIN->
AND NOT   M00619	// L_4th TOOL SD PUNCH FWD/BWD SN ALARM
AND NOT   M11842	// T)4th SIDE PUNCH BWD
OUT       M11634	// L_4th MAND SIDE PUNCH FWD

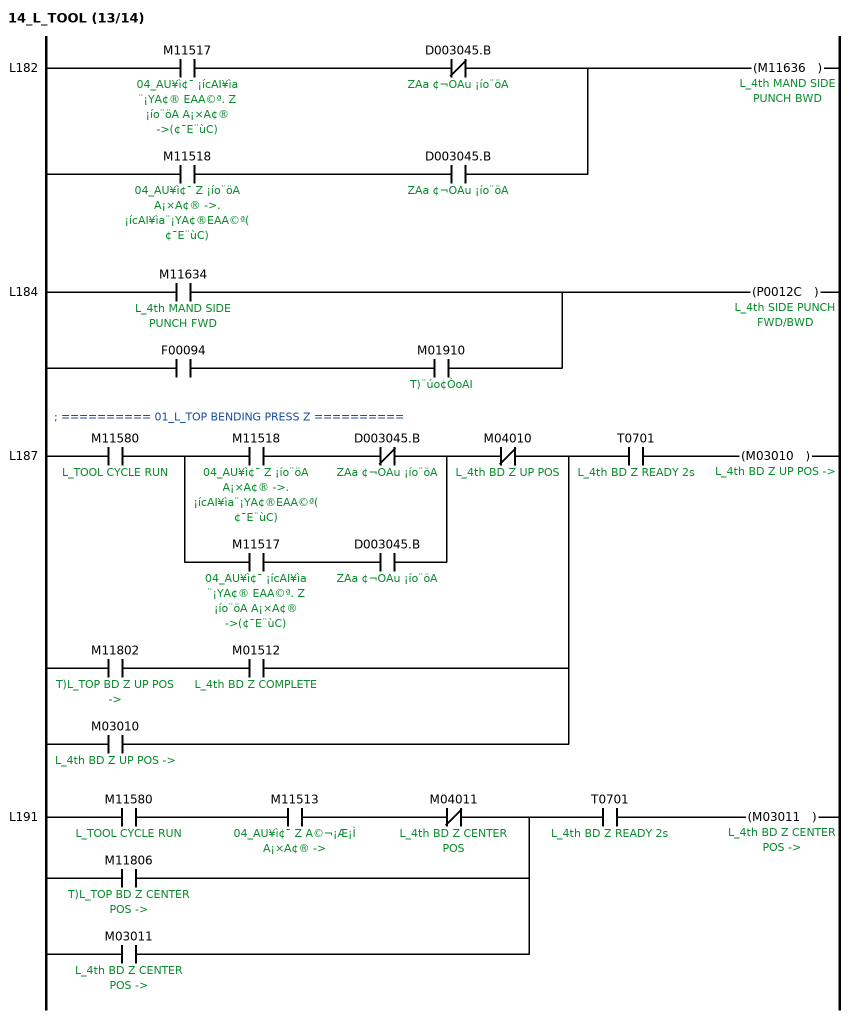
; L182
LOAD      M11517	// 04_AU¥ì¢¯ ¡ícAI¥ìa ¨¡YA¢® EAA©ª. Z ¡ío¨öA A¡×A¢® ->(¢¯E¨ùC)
AND NOT   D003045.B	// ZAa ¢¬OAu ¡ío¨öA
LOAD      M11518	// 04_AU¥ì¢¯ Z ¡ío¨öA A¡×A¢® ->. ¡ícAI¥ìa¨¡YA¢®EAA©ª(¢¯E¨ùC)
AND       D003045.B	// ZAa ¢¬OAu ¡ío¨öA
OR LOAD
OUT       M11636	// L_4th MAND SIDE PUNCH BWD
; L184
LOAD      M11634	// L_4th MAND SIDE PUNCH FWD
LOAD      F00094
AND       M01910	// T)¨úo¢ÒoAI
OR LOAD
OUT       P0012C	// L_4th SIDE PUNCH FWD/BWD
// ========== 01_L_TOP BENDING PRESS Z ==========
; L187
LOAD      M11580	// L_TOOL CYCLE RUN
LOAD      M11518	// 04_AU¥ì¢¯ Z ¡ío¨öA A¡×A¢® ->. ¡ícAI¥ìa¨¡YA¢®EAA©ª(¢¯E¨ùC)
AND NOT   D003045.B	// ZAa ¢¬OAu ¡ío¨öA
LOAD      M11517	// 04_AU¥ì¢¯ ¡ícAI¥ìa ¨¡YA¢® EAA©ª. Z ¡ío¨öA A¡×A¢® ->(¢¯E¨ùC)
AND       D003045.B	// ZAa ¢¬OAu ¡ío¨öA
OR LOAD
AND LOAD
AND NOT   M04010	// L_4th BD Z UP POS
LOAD      M11802	// T)L_TOP BD Z UP POS ->
AND       M01512	// L_4th BD Z COMPLETE
OR LOAD
OR        M03010	// L_4th BD Z UP POS ->
AND       T0701	// L_4th BD Z READY 2s
OUT       M03010	// L_4th BD Z UP POS ->
; L191
LOAD      M11580	// L_TOOL CYCLE RUN
AND       M11513	// 04_AU¥ì¢¯ Z A©¬¡Æ¡Ì A¡×A¢® ->
AND NOT   M04011	// L_4th BD Z CENTER POS
OR        M11806	// T)L_TOP BD Z CENTER POS ->
OR        M03011	// L_4th BD Z CENTER POS ->
AND       T0701	// L_4th BD Z READY 2s
OUT       M03011	// L_4th BD Z CENTER POS ->

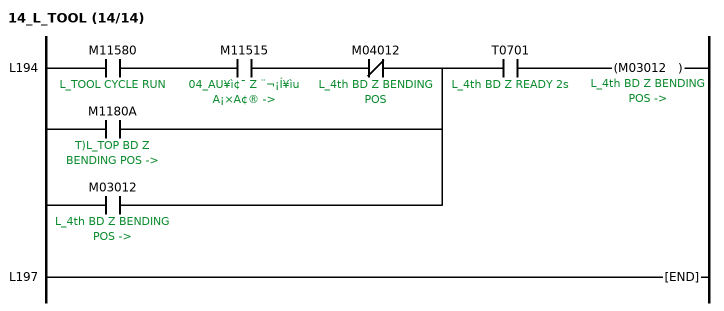
; L194
LOAD      M11580	// L_TOOL CYCLE RUN
AND       M11515	// 04_AU¥ì¢¯ Z ¨¬¡Í¥ìu A¡×A¢® ->
AND NOT   M04012	// L_4th BD Z BENDING POS
OR        M1180A	// T)L_TOP BD Z BENDING POS ->
OR        M03012	// L_4th BD Z BENDING POS ->
AND       T0701	// L_4th BD Z READY 2s
OUT       M03012	// L_4th BD Z BENDING POS ->
; L197
END

PROGRAM 15_L_PP (task: ¨ö¨¬A¥ì CA¡¤I¡¾¡¿¡¤¡Í)

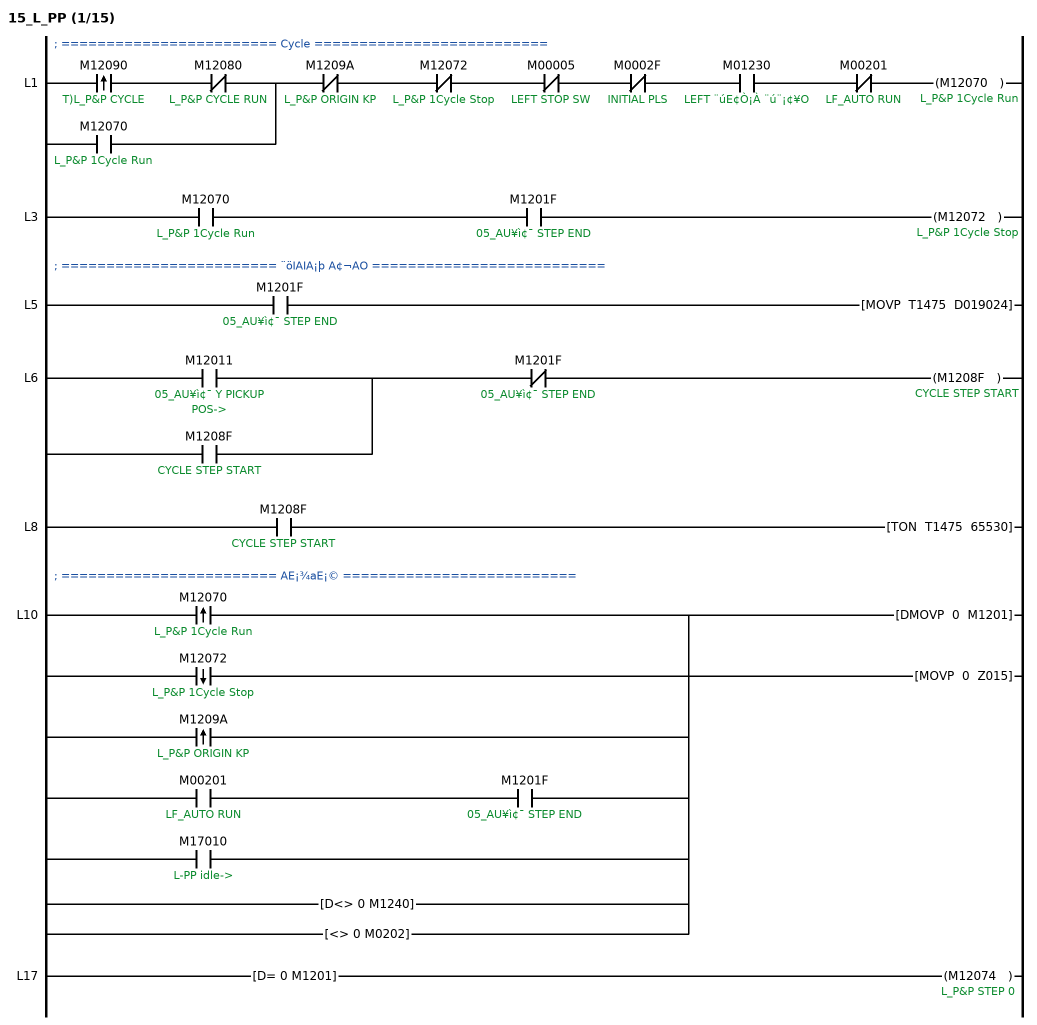
// ======================== Cycle ==========================
; L1
LOADP     M12090	// T)L_P&P CYCLE
AND NOT   M12080	// L_P&P CYCLE RUN
OR        M12070	// L_P&P 1Cycle Run
AND NOT   M1209A	// L_P&P ORIGIN KP
AND NOT   M12072	// L_P&P 1Cycle Stop
AND NOT   M00005	// LEFT STOP SW
AND NOT   M0002F	// INITIAL PLS
AND       M01230	// LEFT ¨úE¢Ò¡À ¨ú¨¡¢¥O
AND NOT   M00201	// LF_AUTO RUN
OUT       M12070	// L_P&P 1Cycle Run
; L3
LOAD      M12070	// L_P&P 1Cycle Run
AND       M1201F	// 05_AU¥ì¢¯ STEP END
OUT       M12072	// L_P&P 1Cycle Stop
// ======================== ¨öIAIA¡þ A¢¬AO ==========================
; L5
LOAD      M1201F	// 05_AU¥ì¢¯ STEP END
MOVP      T1475 D019024
; L6
LOAD      M12011	// 05_AU¥ì¢¯ Y PICKUP POS->
OR        M1208F	// CYCLE STEP START
AND NOT   M1201F	// 05_AU¥ì¢¯ STEP END
OUT       M1208F	// CYCLE STEP START
; L8
LOAD      M1208F	// CYCLE STEP START
TON       T1475 65530
// ======================== AE¡¾aE¡© ==========================
; L10
LOADP     M12070	// L_P&P 1Cycle Run
ORN       M12072	// L_P&P 1Cycle Stop
ORP       M1209A	// L_P&P ORIGIN KP
LOAD      M00201	// LF_AUTO RUN
AND       M1201F	// 05_AU¥ì¢¯ STEP END
OR LOAD
OR        M17010	// L-PP idle->
ORD<>     0 M1240
OR<>      0 M0202
DMOVP     0 M1201
MOVP      0 Z015
; L17
LOADD=    0 M1201
OUT       M12074	// L_P&P STEP 0

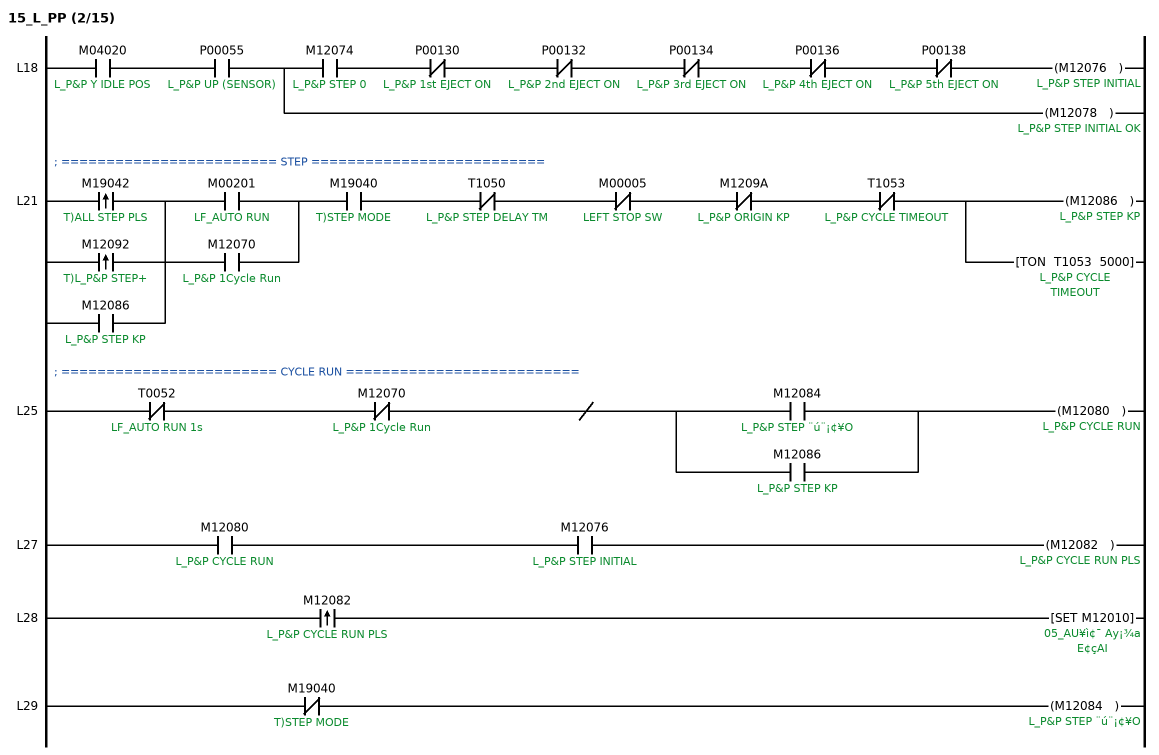
; L18
LOAD      M04020	// L_P&P Y IDLE POS
AND       P00055	// L_P&P UP (SENSOR)
MPUSH
AND       M12074	// L_P&P STEP 0
AND NOT   P00130	// L_P&P 1st EJECT ON
AND NOT   P00132	// L_P&P 2nd EJECT ON
AND NOT   P00134	// L_P&P 3rd EJECT ON
AND NOT   P00136	// L_P&P 4th EJECT ON
AND NOT   P00138	// L_P&P 5th EJECT ON
OUT       M12076	// L_P&P STEP INITIAL
MPOP
OUT       M12078	// L_P&P STEP INITIAL OK
// ======================== STEP ==========================
; L21
LOADP     M19042	// T)ALL STEP PLS
ORP       M12092	// T)L_P&P STEP+
OR        M12086	// L_P&P STEP KP
LOAD      M00201	// LF_AUTO RUN
OR        M12070	// L_P&P 1Cycle Run
AND LOAD
AND       M19040	// T)STEP MODE
AND NOT   T1050	// L_P&P STEP DELAY TM
AND NOT   M00005	// LEFT STOP SW
AND NOT   M1209A	// L_P&P ORIGIN KP
AND NOT   T1053	// L_P&P CYCLE TIMEOUT
OUT       M12086	// L_P&P STEP KP
TON       T1053 5000	// L_P&P CYCLE TIMEOUT
// ======================== CYCLE RUN ==========================
; L25
LOAD NOT  T0052	// LF_AUTO RUN 1s
AND NOT   M12070	// L_P&P 1Cycle Run
NOT
LOAD      M12084	// L_P&P STEP ¨ú¨¡¢¥O
OR        M12086	// L_P&P STEP KP
AND LOAD
OUT       M12080	// L_P&P CYCLE RUN
; L27
LOAD      M12080	// L_P&P CYCLE RUN
AND       M12076	// L_P&P STEP INITIAL
OUT       M12082	// L_P&P CYCLE RUN PLS
; L28
LOADP     M12082	// L_P&P CYCLE RUN PLS
SET       M12010	// 05_AU¥ì¢¯ Ay¡¾a E¢çAI
; L29
LOAD NOT  M19040	// T)STEP MODE
OUT       M12084	// L_P&P STEP ¨ú¨¡¢¥O

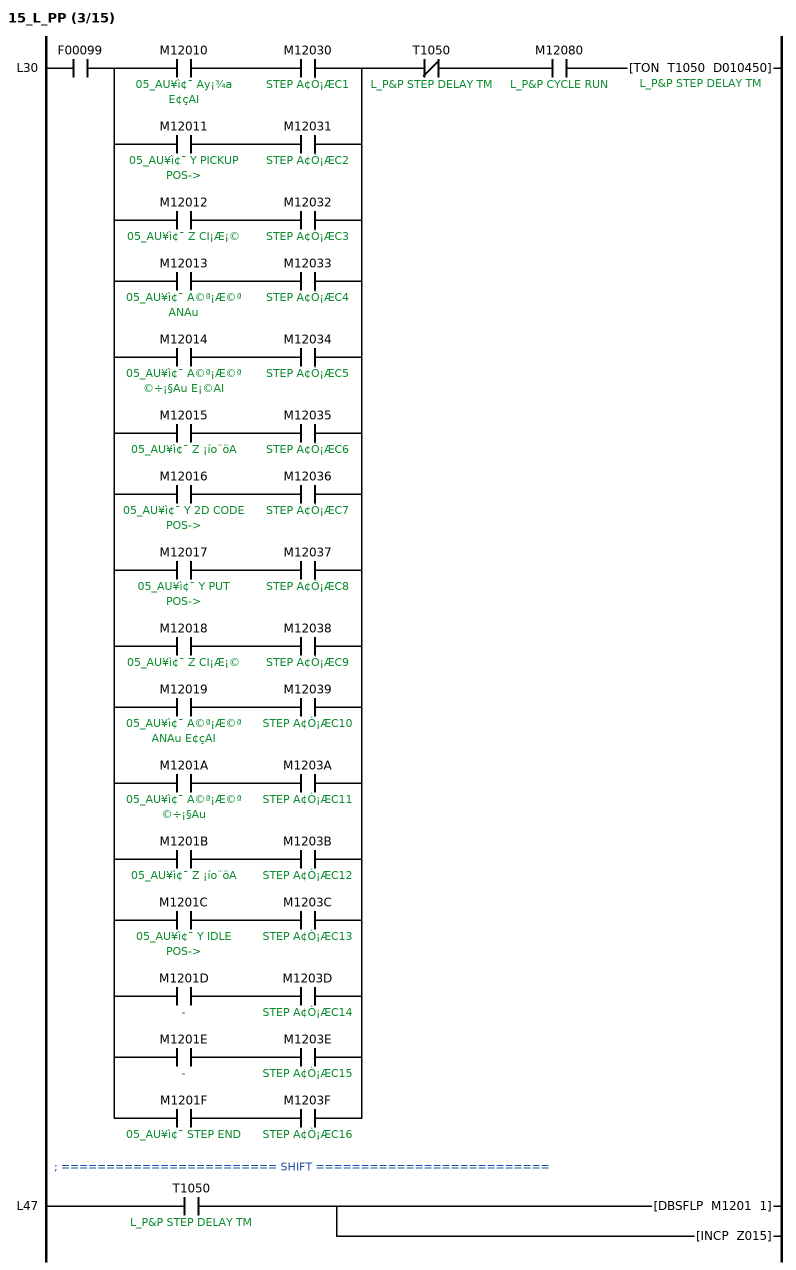
; L30
LOAD      F00099
LOAD      M12010	// 05_AU¥ì¢¯ Ay¡¾a E¢çAI
AND       M12030	// STEP A¢Ò¡ÆC1
LOAD      M12011	// 05_AU¥ì¢¯ Y PICKUP POS->
AND       M12031	// STEP A¢Ò¡ÆC2
OR LOAD
LOAD      M12012	// 05_AU¥ì¢¯ Z CI¡Æ¡©
AND       M12032	// STEP A¢Ò¡ÆC3
OR LOAD
LOAD      M12013	// 05_AU¥ì¢¯ A©ª¡Æ©ª ANAu
AND       M12033	// STEP A¢Ò¡ÆC4
OR LOAD
LOAD      M12014	// 05_AU¥ì¢¯ A©ª¡Æ©ª ©÷¡§Au E¡©AI
AND       M12034	// STEP A¢Ò¡ÆC5
OR LOAD
LOAD      M12015	// 05_AU¥ì¢¯ Z ¡ío¨öA
AND       M12035	// STEP A¢Ò¡ÆC6
OR LOAD
LOAD      M12016	// 05_AU¥ì¢¯ Y 2D CODE POS->
AND       M12036	// STEP A¢Ò¡ÆC7
OR LOAD
LOAD      M12017	// 05_AU¥ì¢¯ Y PUT POS->
AND       M12037	// STEP A¢Ò¡ÆC8
OR LOAD
LOAD      M12018	// 05_AU¥ì¢¯ Z CI¡Æ¡©
AND       M12038	// STEP A¢Ò¡ÆC9
OR LOAD
LOAD      M12019	// 05_AU¥ì¢¯ A©ª¡Æ©ª ANAu E¢çAI
AND       M12039	// STEP A¢Ò¡ÆC10
OR LOAD
LOAD      M1201A	// 05_AU¥ì¢¯ A©ª¡Æ©ª ©÷¡§Au
AND       M1203A	// STEP A¢Ò¡ÆC11
OR LOAD
LOAD      M1201B	// 05_AU¥ì¢¯ Z ¡ío¨öA
AND       M1203B	// STEP A¢Ò¡ÆC12
OR LOAD
LOAD      M1201C	// 05_AU¥ì¢¯ Y IDLE POS->
AND       M1203C	// STEP A¢Ò¡ÆC13
OR LOAD
LOAD      M1201D	// -
AND       M1203D	// STEP A¢Ò¡ÆC14
OR LOAD
LOAD      M1201E	// -
AND       M1203E	// STEP A¢Ò¡ÆC15
OR LOAD
LOAD      M1201F	// 05_AU¥ì¢¯ STEP END
AND       M1203F	// STEP A¢Ò¡ÆC16
OR LOAD
AND LOAD
AND NOT   T1050	// L_P&P STEP DELAY TM
AND       M12080	// L_P&P CYCLE RUN
TON       T1050 D010450	// L_P&P STEP DELAY TM
// ======================== SHIFT ==========================
; L47
LOAD      T1050	// L_P&P STEP DELAY TM
DBSFLP    M1201 1
INCP      Z015

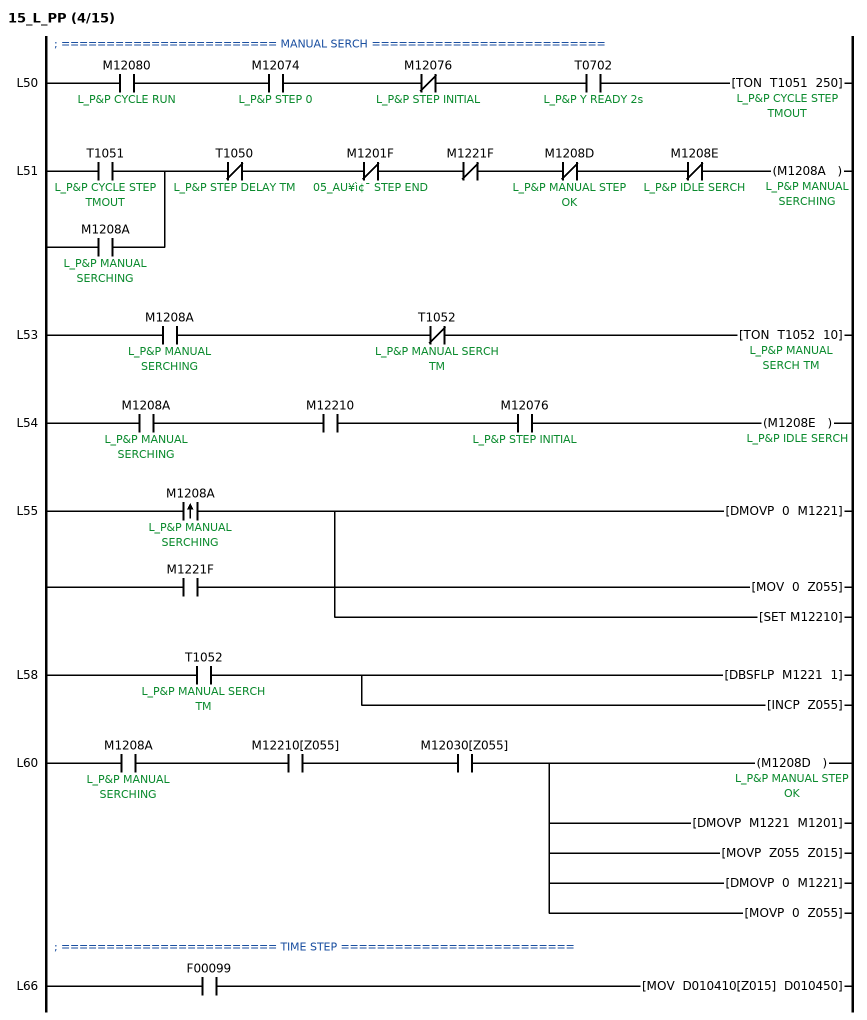
// ======================== MANUAL SERCH ==========================
; L50
LOAD      M12080	// L_P&P CYCLE RUN
AND       M12074	// L_P&P STEP 0
AND NOT   M12076	// L_P&P STEP INITIAL
AND       T0702	// L_P&P Y READY 2s
TON       T1051 250	// L_P&P CYCLE STEP TMOUT
; L51
LOAD      T1051	// L_P&P CYCLE STEP TMOUT
OR        M1208A	// L_P&P MANUAL SERCHING
AND NOT   T1050	// L_P&P STEP DELAY TM
AND NOT   M1201F	// 05_AU¥ì¢¯ STEP END
AND NOT   M1221F
AND NOT   M1208D	// L_P&P MANUAL STEP OK
AND NOT   M1208E	// L_P&P IDLE SERCH
OUT       M1208A	// L_P&P MANUAL SERCHING
; L53
LOAD      M1208A	// L_P&P MANUAL SERCHING
AND NOT   T1052	// L_P&P MANUAL SERCH TM
TON       T1052 10	// L_P&P MANUAL SERCH TM
; L54
LOAD      M1208A	// L_P&P MANUAL SERCHING
AND       M12210
AND       M12076	// L_P&P STEP INITIAL
OUT       M1208E	// L_P&P IDLE SERCH
; L55
LOADP     M1208A	// L_P&P MANUAL SERCHING
OR        M1221F
DMOVP     0 M1221
MOV       0 Z055
SET       M12210
; L58
LOAD      T1052	// L_P&P MANUAL SERCH TM
DBSFLP    M1221 1
INCP      Z055
; L60
LOAD      M1208A	// L_P&P MANUAL SERCHING
AND       M12210[Z055]
AND       M12030[Z055]
OUT       M1208D	// L_P&P MANUAL STEP OK
DMOVP     M1221 M1201
MOVP      Z055 Z015
DMOVP     0 M1221
MOVP      0 Z055
// ======================== TIME STEP ==========================
; L66
LOAD      F00099
MOV       D010410[Z015] D010450

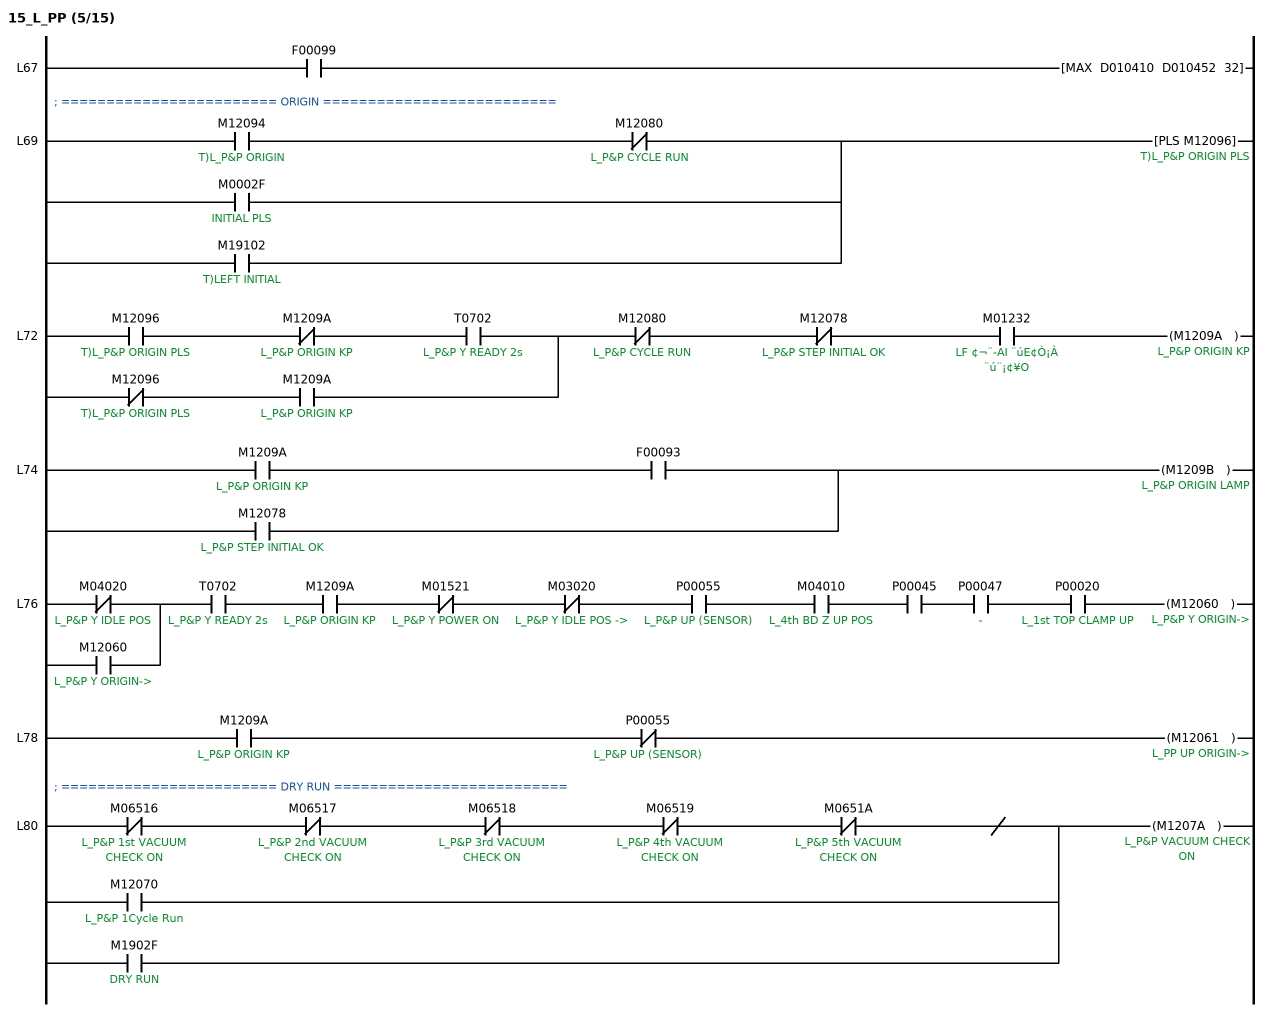
; L67
LOAD      F00099
MAX       D010410 D010452 32
// ======================== ORIGIN ==========================
; L69
LOAD      M12094	// T)L_P&P ORIGIN
AND NOT   M12080	// L_P&P CYCLE RUN
OR        M0002F	// INITIAL PLS
OR        M19102	// T)LEFT INITIAL
OUTP      M12096	// T)L_P&P ORIGIN PLS
; L72
LOAD      M12096	// T)L_P&P ORIGIN PLS
AND NOT   M1209A	// L_P&P ORIGIN KP
AND       T0702	// L_P&P Y READY 2s
LOAD NOT  M12096	// T)L_P&P ORIGIN PLS
AND       M1209A	// L_P&P ORIGIN KP
OR LOAD
AND NOT   M12080	// L_P&P CYCLE RUN
AND NOT   M12078	// L_P&P STEP INITIAL OK
AND       M01232	// LF ¢¬¨­AI ¨úE¢Ò¡À ¨ú¨¡¢¥O
OUT       M1209A	// L_P&P ORIGIN KP
; L74
LOAD      M1209A	// L_P&P ORIGIN KP
AND       F00093
OR        M12078	// L_P&P STEP INITIAL OK
OUT       M1209B	// L_P&P ORIGIN LAMP
; L76
LOAD NOT  M04020	// L_P&P Y IDLE POS
OR        M12060	// L_P&P Y ORIGIN->
AND       T0702	// L_P&P Y READY 2s
AND       M1209A	// L_P&P ORIGIN KP
AND NOT   M01521	// L_P&P Y POWER ON
AND NOT   M03020	// L_P&P Y IDLE POS ->
AND       P00055	// L_P&P UP (SENSOR)
AND       M04010	// L_4th BD Z UP POS
AND       P00045
AND       P00047	// -
AND       P00020	// L_1st TOP CLAMP UP
OUT       M12060	// L_P&P Y ORIGIN->
; L78
LOAD      M1209A	// L_P&P ORIGIN KP
AND NOT   P00055	// L_P&P UP (SENSOR)
OUT       M12061	// L_PP UP ORIGIN->
// ======================== DRY RUN ==========================
; L80
LOAD NOT  M06516	// L_P&P 1st VACUUM CHECK ON
AND NOT   M06517	// L_P&P 2nd VACUUM CHECK ON
AND NOT   M06518	// L_P&P 3rd VACUUM CHECK ON
AND NOT   M06519	// L_P&P 4th VACUUM CHECK ON
AND NOT   M0651A	// L_P&P 5th VACUUM CHECK ON
NOT
OR        M12070	// L_P&P 1Cycle Run
OR        M1902F	// DRY RUN
OUT       M1207A	// L_P&P VACUUM CHECK ON

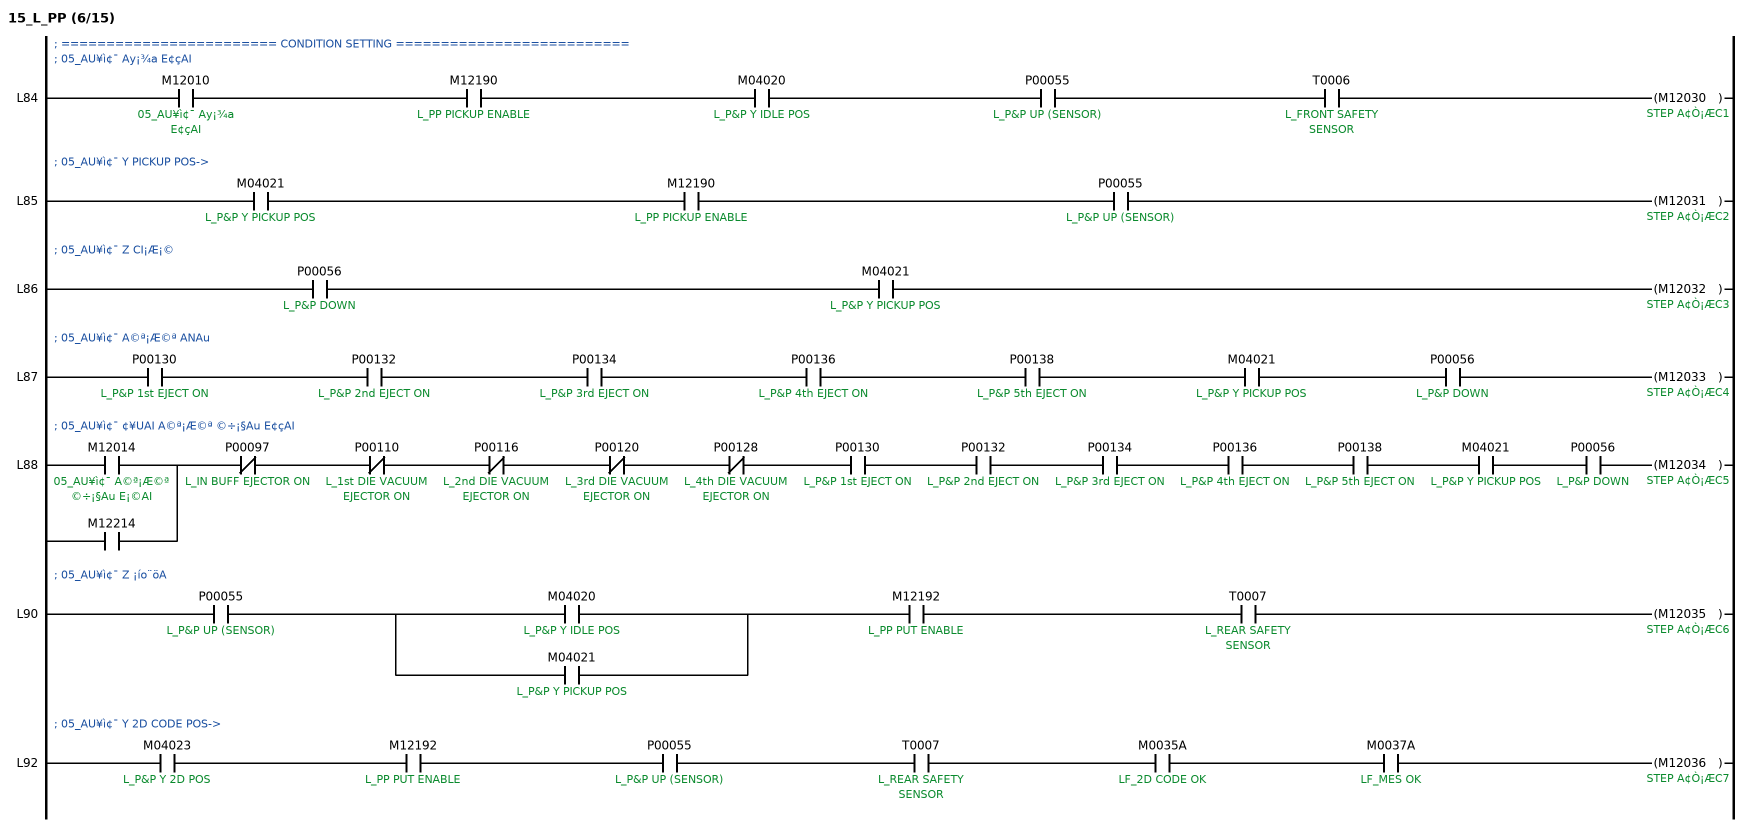
// ======================== CONDITION SETTING ==========================
; L84
LOAD      M12010	// 05_AU¥ì¢¯ Ay¡¾a E¢çAI
AND       M12190	// L_PP PICKUP ENABLE
AND       M04020	// L_P&P Y IDLE POS
AND       P00055	// L_P&P UP (SENSOR)
AND       T0006	// L_FRONT SAFETY SENSOR
OUT       M12030	// STEP A¢Ò¡ÆC1
// output comment: 05_AU¥ì¢¯ Ay¡¾a E¢çAI
; L85
LOAD      M04021	// L_P&P Y PICKUP POS
AND       M12190	// L_PP PICKUP ENABLE
AND       P00055	// L_P&P UP (SENSOR)
OUT       M12031	// STEP A¢Ò¡ÆC2
// output comment: 05_AU¥ì¢¯ Y PICKUP POS->
; L86
LOAD      P00056	// L_P&P DOWN
AND       M04021	// L_P&P Y PICKUP POS
OUT       M12032	// STEP A¢Ò¡ÆC3
// output comment: 05_AU¥ì¢¯ Z CI¡Æ¡©
; L87
LOAD      P00130	// L_P&P 1st EJECT ON
AND       P00132	// L_P&P 2nd EJECT ON
AND       P00134	// L_P&P 3rd EJECT ON
AND       P00136	// L_P&P 4th EJECT ON
AND       P00138	// L_P&P 5th EJECT ON
AND       M04021	// L_P&P Y PICKUP POS
AND       P00056	// L_P&P DOWN
OUT       M12033	// STEP A¢Ò¡ÆC4
// output comment: 05_AU¥ì¢¯ A©ª¡Æ©ª ANAu
; L88
LOAD      M12014	// 05_AU¥ì¢¯ A©ª¡Æ©ª ©÷¡§Au E¡©AI
OR        M12214
AND NOT   P00097	// L_IN BUFF EJECTOR ON
AND NOT   P00110	// L_1st DIE VACUUM EJECTOR ON
AND NOT   P00116	// L_2nd DIE VACUUM EJECTOR ON
AND NOT   P00120	// L_3rd DIE VACUUM EJECTOR ON
AND NOT   P00128	// L_4th DIE VACUUM EJECTOR ON
AND       P00130	// L_P&P 1st EJECT ON
AND       P00132	// L_P&P 2nd EJECT ON
AND       P00134	// L_P&P 3rd EJECT ON
AND       P00136	// L_P&P 4th EJECT ON
AND       P00138	// L_P&P 5th EJECT ON
AND       M04021	// L_P&P Y PICKUP POS
AND       P00056	// L_P&P DOWN
OUT       M12034	// STEP A¢Ò¡ÆC5
// output comment: 05_AU¥ì¢¯ ¢¥UAI A©ª¡Æ©ª ©÷¡§Au E¢çAI
; L90
LOAD      P00055	// L_P&P UP (SENSOR)
LOAD      M04020	// L_P&P Y IDLE POS
OR        M04021	// L_P&P Y PICKUP POS
AND LOAD
AND       M12192	// L_PP PUT ENABLE
AND       T0007	// L_REAR SAFETY SENSOR
OUT       M12035	// STEP A¢Ò¡ÆC6
// output comment: 05_AU¥ì¢¯ Z ¡ío¨öA
; L92
LOAD      M04023	// L_P&P Y 2D POS
AND       M12192	// L_PP PUT ENABLE
AND       P00055	// L_P&P UP (SENSOR)
AND       T0007	// L_REAR SAFETY SENSOR
AND       M0035A	// LF_2D CODE OK
AND       M0037A	// LF_MES OK
OUT       M12036	// STEP A¢Ò¡ÆC7
// output comment: 05_AU¥ì¢¯ Y 2D CODE POS->

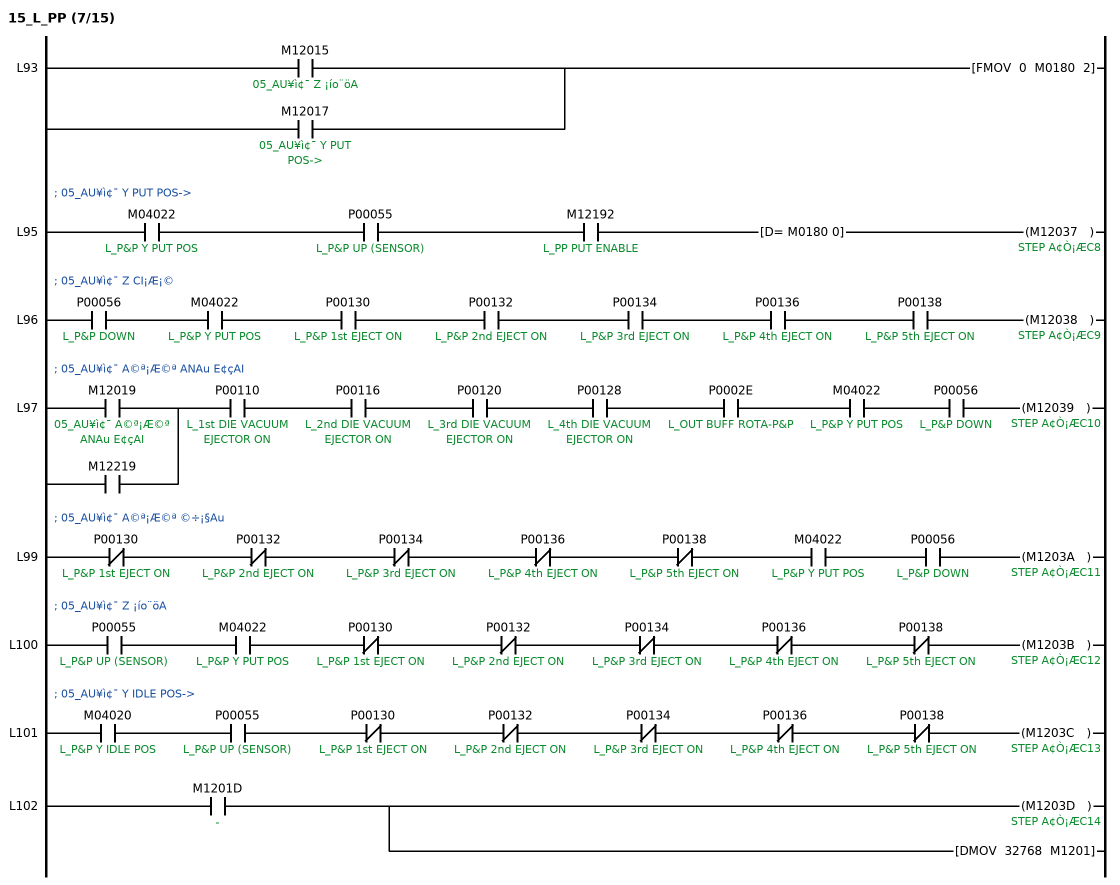
; L93
LOAD      M12015	// 05_AU¥ì¢¯ Z ¡ío¨öA
OR        M12017	// 05_AU¥ì¢¯ Y PUT POS->
FMOV      0 M0180 2
; L95
LOAD      M04022	// L_P&P Y PUT POS
AND       P00055	// L_P&P UP (SENSOR)
AND       M12192	// L_PP PUT ENABLE
ANDD=     M0180 0
OUT       M12037	// STEP A¢Ò¡ÆC8
// output comment: 05_AU¥ì¢¯ Y PUT POS->
; L96
LOAD      P00056	// L_P&P DOWN
AND       M04022	// L_P&P Y PUT POS
AND       P00130	// L_P&P 1st EJECT ON
AND       P00132	// L_P&P 2nd EJECT ON
AND       P00134	// L_P&P 3rd EJECT ON
AND       P00136	// L_P&P 4th EJECT ON
AND       P00138	// L_P&P 5th EJECT ON
OUT       M12038	// STEP A¢Ò¡ÆC9
// output comment: 05_AU¥ì¢¯ Z CI¡Æ¡©
; L97
LOAD      M12019	// 05_AU¥ì¢¯ A©ª¡Æ©ª ANAu E¢çAI
OR        M12219
AND       P00110	// L_1st DIE VACUUM EJECTOR ON
AND       P00116	// L_2nd DIE VACUUM EJECTOR ON
AND       P00120	// L_3rd DIE VACUUM EJECTOR ON
AND       P00128	// L_4th DIE VACUUM EJECTOR ON
AND       P0002E	// L_OUT BUFF ROTA-P&P
AND       M04022	// L_P&P Y PUT POS
AND       P00056	// L_P&P DOWN
OUT       M12039	// STEP A¢Ò¡ÆC10
// output comment: 05_AU¥ì¢¯ A©ª¡Æ©ª ANAu E¢çAI
; L99
LOAD NOT  P00130	// L_P&P 1st EJECT ON
AND NOT   P00132	// L_P&P 2nd EJECT ON
AND NOT   P00134	// L_P&P 3rd EJECT ON
AND NOT   P00136	// L_P&P 4th EJECT ON
AND NOT   P00138	// L_P&P 5th EJECT ON
AND       M04022	// L_P&P Y PUT POS
AND       P00056	// L_P&P DOWN
OUT       M1203A	// STEP A¢Ò¡ÆC11
// output comment: 05_AU¥ì¢¯ A©ª¡Æ©ª ©÷¡§Au
; L100
LOAD      P00055	// L_P&P UP (SENSOR)
AND       M04022	// L_P&P Y PUT POS
AND NOT   P00130	// L_P&P 1st EJECT ON
AND NOT   P00132	// L_P&P 2nd EJECT ON
AND NOT   P00134	// L_P&P 3rd EJECT ON
AND NOT   P00136	// L_P&P 4th EJECT ON
AND NOT   P00138	// L_P&P 5th EJECT ON
OUT       M1203B	// STEP A¢Ò¡ÆC12
// output comment: 05_AU¥ì¢¯ Z ¡ío¨öA
; L101
LOAD      M04020	// L_P&P Y IDLE POS
AND       P00055	// L_P&P UP (SENSOR)
AND NOT   P00130	// L_P&P 1st EJECT ON
AND NOT   P00132	// L_P&P 2nd EJECT ON
AND NOT   P00134	// L_P&P 3rd EJECT ON
AND NOT   P00136	// L_P&P 4th EJECT ON
AND NOT   P00138	// L_P&P 5th EJECT ON
OUT       M1203C	// STEP A¢Ò¡ÆC13
// output comment: 05_AU¥ì¢¯ Y IDLE POS->
; L102
LOAD      M1201D	// -
OUT       M1203D	// STEP A¢Ò¡ÆC14
DMOV      32768 M1201

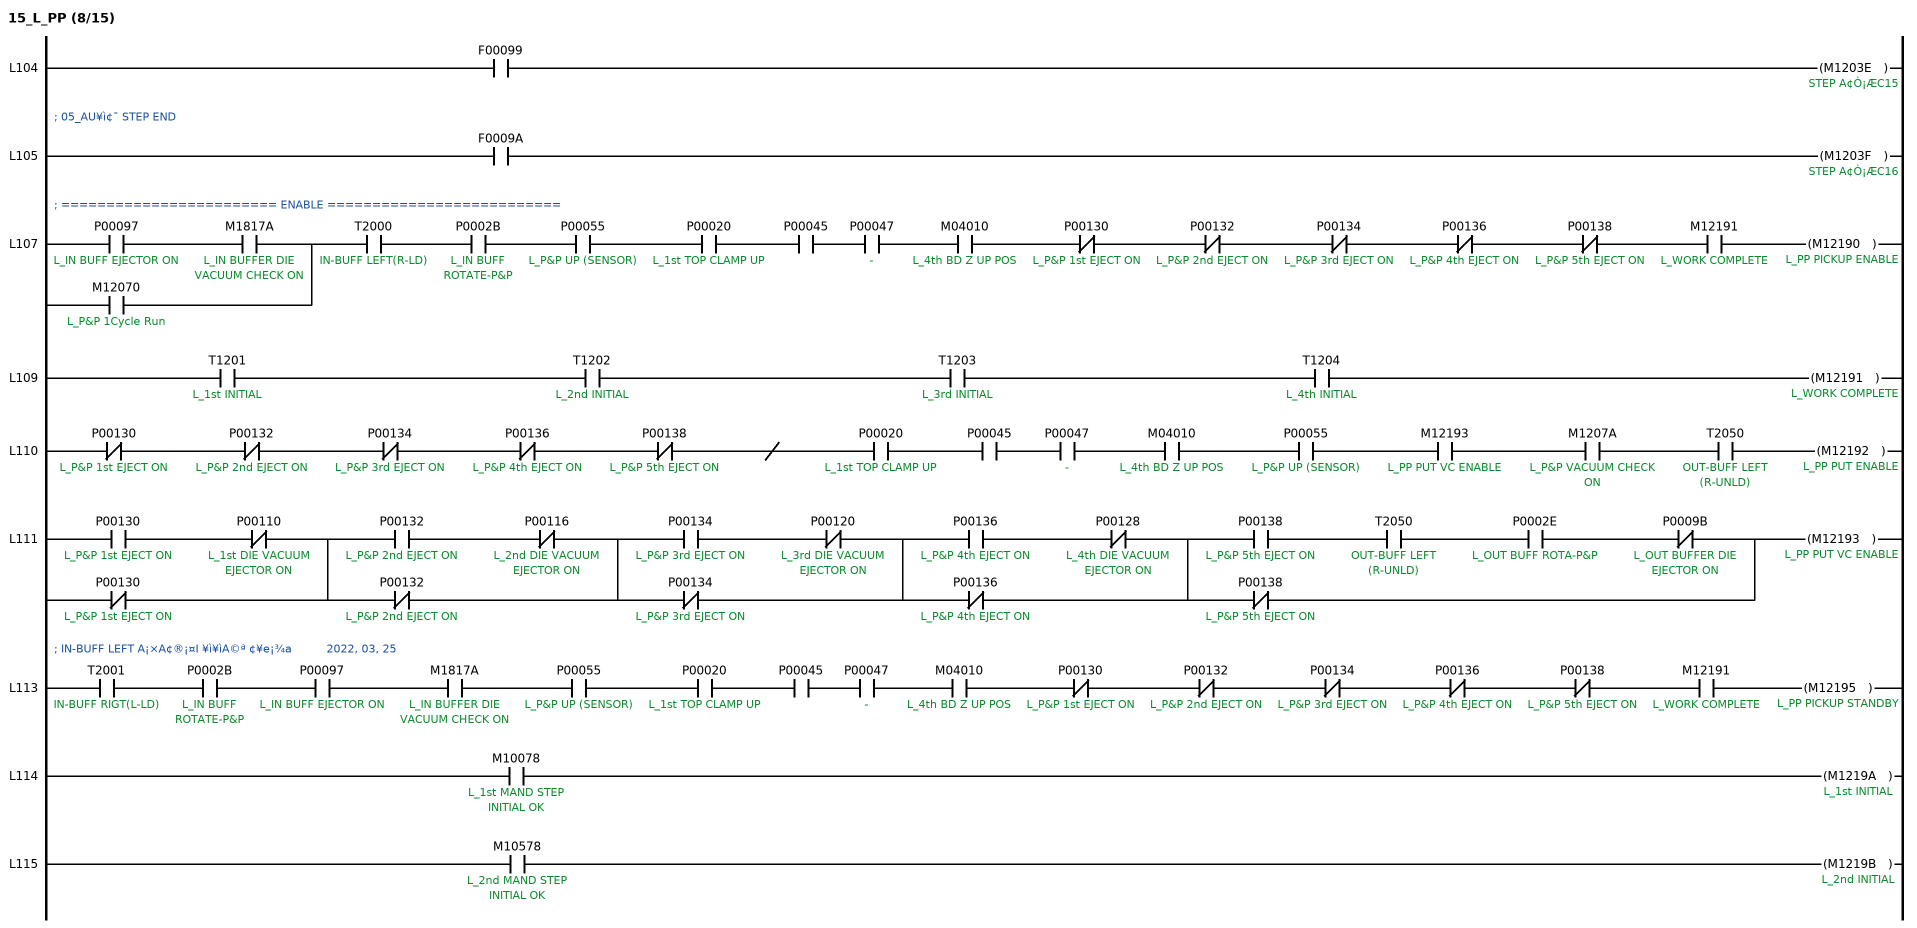
; L104
LOAD      F00099
OUT       M1203E	// STEP A¢Ò¡ÆC15
; L105
LOAD      F0009A
OUT       M1203F	// STEP A¢Ò¡ÆC16
// output comment: 05_AU¥ì¢¯ STEP END
// ======================== ENABLE ==========================
; L107
LOAD      P00097	// L_IN BUFF EJECTOR ON
AND       M1817A	// L_IN BUFFER DIE VACUUM CHECK ON
OR        M12070	// L_P&P 1Cycle Run
AND       T2000	// IN-BUFF LEFT(R-LD)
AND       P0002B	// L_IN BUFF ROTATE-P&P
AND       P00055	// L_P&P UP (SENSOR)
AND       P00020	// L_1st TOP CLAMP UP
AND       P00045
AND       P00047	// -
AND       M04010	// L_4th BD Z UP POS
AND NOT   P00130	// L_P&P 1st EJECT ON
AND NOT   P00132	// L_P&P 2nd EJECT ON
AND NOT   P00134	// L_P&P 3rd EJECT ON
AND NOT   P00136	// L_P&P 4th EJECT ON
AND NOT   P00138	// L_P&P 5th EJECT ON
AND       M12191	// L_WORK COMPLETE
OUT       M12190	// L_PP PICKUP ENABLE
; L109
LOAD      T1201	// L_1st INITIAL
AND       T1202	// L_2nd INITIAL
AND       T1203	// L_3rd INITIAL
AND       T1204	// L_4th INITIAL
OUT       M12191	// L_WORK COMPLETE
; L110
LOAD NOT  P00130	// L_P&P 1st EJECT ON
AND NOT   P00132	// L_P&P 2nd EJECT ON
AND NOT   P00134	// L_P&P 3rd EJECT ON
AND NOT   P00136	// L_P&P 4th EJECT ON
AND NOT   P00138	// L_P&P 5th EJECT ON
NOT
AND       P00020	// L_1st TOP CLAMP UP
AND       P00045
AND       P00047	// -
AND       M04010	// L_4th BD Z UP POS
AND       P00055	// L_P&P UP (SENSOR)
AND       M12193	// L_PP PUT VC ENABLE
AND       M1207A	// L_P&P VACUUM CHECK ON
AND       T2050	// OUT-BUFF LEFT (R-UNLD)
OUT       M12192	// L_PP PUT ENABLE
; L111
LOAD      P00130	// L_P&P 1st EJECT ON
AND NOT   P00110	// L_1st DIE VACUUM EJECTOR ON
OR NOT    P00130	// L_P&P 1st EJECT ON
LOAD      P00132	// L_P&P 2nd EJECT ON
AND NOT   P00116	// L_2nd DIE VACUUM EJECTOR ON
OR NOT    P00132	// L_P&P 2nd EJECT ON
AND LOAD
LOAD      P00134	// L_P&P 3rd EJECT ON
AND NOT   P00120	// L_3rd DIE VACUUM EJECTOR ON
OR NOT    P00134	// L_P&P 3rd EJECT ON
AND LOAD
LOAD      P00136	// L_P&P 4th EJECT ON
AND NOT   P00128	// L_4th DIE VACUUM EJECTOR ON
OR NOT    P00136	// L_P&P 4th EJECT ON
AND LOAD
LOAD      P00138	// L_P&P 5th EJECT ON
AND       T2050	// OUT-BUFF LEFT (R-UNLD)
AND       P0002E	// L_OUT BUFF ROTA-P&P
AND NOT   P0009B	// L_OUT BUFFER DIE EJECTOR ON
OR NOT    P00138	// L_P&P 5th EJECT ON
AND LOAD
OUT       M12193	// L_PP PUT VC ENABLE
; L113
LOAD      T2001	// IN-BUFF RIGT(L-LD)
AND       P0002B	// L_IN BUFF ROTATE-P&P
AND       P00097	// L_IN BUFF EJECTOR ON
AND       M1817A	// L_IN BUFFER DIE VACUUM CHECK ON
AND       P00055	// L_P&P UP (SENSOR)
AND       P00020	// L_1st TOP CLAMP UP
AND       P00045
AND       P00047	// -
AND       M04010	// L_4th BD Z UP POS
AND NOT   P00130	// L_P&P 1st EJECT ON
AND NOT   P00132	// L_P&P 2nd EJECT ON
AND NOT   P00134	// L_P&P 3rd EJECT ON
AND NOT   P00136	// L_P&P 4th EJECT ON
AND NOT   P00138	// L_P&P 5th EJECT ON
AND       M12191	// L_WORK COMPLETE
OUT       M12195	// L_PP PICKUP STANDBY
// output comment: IN-BUFF LEFT A¡×A¢®¡¤I ¥ì¥ìA©ª ¢¥e¡¾a          2022, 03, 25
; L114
LOAD      M10078	// L_1st MAND STEP INITIAL OK
OUT       M1219A	// L_1st INITIAL
; L115
LOAD      M10578	// L_2nd MAND STEP INITIAL OK
OUT       M1219B	// L_2nd INITIAL

